//     PlcTask Inputs/GVL_iXlinker.EtherCAT_Master_EPPxxxx.Beckhoff_EPP6xxx.Beckhoff_EPP6xxxEK1122.A_0002_EPP6001_0002_0017.COM_Inputs.Data_In[11] <-> COM Inputs/Data In 11
//     PlcTask Inputs/GVL_iXlinker.EtherCAT_Master_EPPxxxx.Beckhoff_EPP6xxx.Beckhoff_EPP6xxxEK1122.A_0002_EPP6001_0002_0017.COM_Inputs.Data_In[12] <-> COM Inputs/Data In 12
//     PlcTask Inputs/GVL_iXlinker.EtherCAT_Master_EPPxxxx.Beckhoff_EPP6xxx.Beckhoff_EPP6xxxEK1122.A_0002_EPP6001_0002_0017.COM_Inputs.Data_In[13] <-> COM Inputs/Data In 13
//     PlcTask Inputs/GVL_iXlinker.EtherCAT_Master_EPPxxxx.Beckhoff_EPP6xxx.Beckhoff_EPP6xxxEK1122.A_0002_EPP6001_0002_0017.COM_Inputs.Data_In[14] <-> COM Inputs/Data In 14
//     PlcTask Inputs/GVL_iXlinker.EtherCAT_Master_EPPxxxx.Beckhoff_EPP6xxx.Beckhoff_EPP6xxxEK1122.A_0002_EPP6001_0002_0017.COM_Inputs.Data_In[15] <-> COM Inputs/Data In 15
//     PlcTask Inputs/GVL_iXlinker.EtherCAT_Master_EPPxxxx.Beckhoff_EPP6xxx.Beckhoff_EPP6xxxEK1122.A_0002_EPP6001_0002_0017.COM_Inputs.Data_In[16] <-> COM Inputs/Data In 16
//     PlcTask Inputs/GVL_iXlinker.EtherCAT_Master_EPPxxxx.Beckhoff_EPP6xxx.Beckhoff_EPP6xxxEK1122.A_0002_EPP6001_0002_0017.COM_Inputs.Data_In[17] <-> COM Inputs/Data In 17
//     PlcTask Inputs/GVL_iXlinker.EtherCAT_Master_EPPxxxx.Beckhoff_EPP6xxx.Beckhoff_EPP6xxxEK1122.A_0002_EPP6001_0002_0017.COM_Inputs.Data_In[18] <-> COM Inputs/Data In 18
//     PlcTask Inputs/GVL_iXlinker.EtherCAT_Master_EPPxxxx.Beckhoff_EPP6xxx.Beckhoff_EPP6xxxEK1122.A_0002_EPP6001_0002_0017.COM_Inputs.Data_In[19] <-> COM Inputs/Data In 19
//     PlcTask Inputs/GVL_iXlinker.EtherCAT_Master_EPPxxxx.Beckhoff_EPP6xxx.Beckhoff_EPP6xxxEK1122.A_0002_EPP6001_0002_0017.COM_Inputs.Data_In[20] <-> COM Inputs/Data In 20
//     PlcTask Inputs/GVL_iXlinker.EtherCAT_Master_EPPxxxx.Beckhoff_EPP6xxx.Beckhoff_EPP6xxxEK1122.A_0002_EPP6001_0002_0017.COM_Inputs.Data_In[21] <-> COM Inputs/Data In 21
//     PlcTask Outputs/GVL_iXlinker.EtherCAT_Master_EPPxxxx.Beckhoff_EPP6xxx.Beckhoff_EPP6xxxEK1122.A_0002_EPP6001_0002_0017.COM_Outputs.Ctrl <-> COM Outputs/Ctrl
//     PlcTask Outputs/GVL_iXlinker.EtherCAT_Master_EPPxxxx.Beckhoff_EPP6xxx.Beckhoff_EPP6xxxEK1122.A_0002_EPP6001_0002_0017.COM_Outputs.Data_Out[0] <-> COM Outputs/Data Out 0
//     PlcTask Outputs/GVL_iXlinker.EtherCAT_Master_EPPxxxx.Beckhoff_EPP6xxx.Beckhoff_EPP6xxxEK1122.A_0002_EPP6001_0002_0017.COM_Outputs.Data_Out[1] <-> COM Outputs/Data Out 1
//     PlcTask Outputs/GVL_iXlinker.EtherCAT_Master_EPPxxxx.Beckhoff_EPP6xxx.Beckhoff_EPP6xxxEK1122.A_0002_EPP6001_0002_0017.COM_Outputs.Data_Out[2] <-> COM Outputs/Data Out 2
//     PlcTask Outputs/GVL_iXlinker.EtherCAT_Master_EPPxxxx.Beckhoff_EPP6xxx.Beckhoff_EPP6xxxEK1122.A_0002_EPP6001_0002_0017.COM_Outputs.Data_Out[3] <-> COM Outputs/Data Out 3
//     PlcTask Outputs/GVL_iXlinker.EtherCAT_Master_EPPxxxx.Beckhoff_EPP6xxx.Beckhoff_EPP6xxxEK1122.A_0002_EPP6001_0002_0017.COM_Outputs.Data_Out[4] <-> COM Outputs/Data Out 4
//     PlcTask Outputs/GVL_iXlinker.EtherCAT_Master_EPPxxxx.Beckhoff_EPP6xxx.Beckhoff_EPP6xxxEK1122.A_0002_EPP6001_0002_0017.COM_Outputs.Data_Out[5] <-> COM Outputs/Data Out 5
//     PlcTask Outputs/GVL_iXlinker.EtherCAT_Master_EPPxxxx.Beckhoff_EPP6xxx.Beckhoff_EPP6xxxEK1122.A_0002_EPP6001_0002_0017.COM_Outputs.Data_Out[6] <-> COM Outputs/Data Out 6
//     PlcTask Outputs/GVL_iXlinker.EtherCAT_Master_EPPxxxx.Beckhoff_EPP6xxx.Beckhoff_EPP6xxxEK1122.A_0002_EPP6001_0002_0017.COM_Outputs.Data_Out[7] <-> COM Outputs/Data Out 7
//     PlcTask Outputs/GVL_iXlinker.EtherCAT_Master_EPPxxxx.Beckhoff_EPP6xxx.Beckhoff_EPP6xxxEK1122.A_0002_EPP6001_0002_0017.COM_Outputs.Data_Out[8] <-> COM Outputs/Data Out 8
//     PlcTask Outputs/GVL_iXlinker.EtherCAT_Master_EPPxxxx.Beckhoff_EPP6xxx.Beckhoff_EPP6xxxEK1122.A_0002_EPP6001_0002_0017.COM_Outputs.Data_Out[9] <-> COM Outputs/Data Out 9
//     PlcTask Outputs/GVL_iXlinker.EtherCAT_Master_EPPxxxx.Beckhoff_EPP6xxx.Beckhoff_EPP6xxxEK1122.A_0002_EPP6001_0002_0017.COM_Outputs.Data_Out[10] <-> COM Outputs/Data Out 10
//     PlcTask Outputs/GVL_iXlinker.EtherCAT_Master_EPPxxxx.Beckhoff_EPP6xxx.Beckhoff_EPP6xxxEK1122.A_0002_EPP6001_0002_0017.COM_Outputs.Data_Out[11] <-> COM Outputs/Data Out 11
//     PlcTask Outputs/GVL_iXlinker.EtherCAT_Master_EPPxxxx.Beckhoff_EPP6xxx.Beckhoff_EPP6xxxEK1122.A_0002_EPP6001_0002_0017.COM_Outputs.Data_Out[12] <-> COM Outputs/Data Out 12
//     PlcTask Outputs/GVL_iXlinker.EtherCAT_Master_EPPxxxx.Beckhoff_EPP6xxx.Beckhoff_EPP6xxxEK1122.A_0002_EPP6001_0002_0017.COM_Outputs.Data_Out[13] <-> COM Outputs/Data Out 13
//     PlcTask Outputs/GVL_iXlinker.EtherCAT_Master_EPPxxxx.Beckhoff_EPP6xxx.Beckhoff_EPP6xxxEK1122.A_0002_EPP6001_0002_0017.COM_Outputs.Data_Out[14] <-> COM Outputs/Data Out 14
//     PlcTask Outputs/GVL_iXlinker.EtherCAT_Master_EPPxxxx.Beckhoff_EPP6xxx.Beckhoff_EPP6xxxEK1122.A_0002_EPP6001_0002_0017.COM_Outputs.Data_Out[15] <-> COM Outputs/Data Out 15
//     PlcTask Outputs/GVL_iXlinker.EtherCAT_Master_EPPxxxx.Beckhoff_EPP6xxx.Beckhoff_EPP6xxxEK1122.A_0002_EPP6001_0002_0017.COM_Outputs.Data_Out[16] <-> COM Outputs/Data Out 16
//     PlcTask Outputs/GVL_iXlinker.EtherCAT_Master_EPPxxxx.Beckhoff_EPP6xxx.Beckhoff_EPP6xxxEK1122.A_0002_EPP6001_0002_0017.COM_Outputs.Data_Out[17] <-> COM Outputs/Data Out 17
//     PlcTask Outputs/GVL_iXlinker.EtherCAT_Master_EPPxxxx.Beckhoff_EPP6xxx.Beckhoff_EPP6xxxEK1122.A_0002_EPP6001_0002_0017.COM_Outputs.Data_Out[18] <-> COM Outputs/Data Out 18
//     PlcTask Outputs/GVL_iXlinker.EtherCAT_Master_EPPxxxx.Beckhoff_EPP6xxx.Beckhoff_EPP6xxxEK1122.A_0002_EPP6001_0002_0017.COM_Outputs.Data_Out[19] <-> COM Outputs/Data Out 19
//     PlcTask Outputs/GVL_iXlinker.EtherCAT_Master_EPPxxxx.Beckhoff_EPP6xxx.Beckhoff_EPP6xxxEK1122.A_0002_EPP6001_0002_0017.COM_Outputs.Data_Out[20] <-> COM Outputs/Data Out 20
//     PlcTask Outputs/GVL_iXlinker.EtherCAT_Master_EPPxxxx.Beckhoff_EPP6xxx.Beckhoff_EPP6xxxEK1122.A_0002_EPP6001_0002_0017.COM_Outputs.Data_Out[21] <-> COM Outputs/Data Out 21
//     PlcTask Inputs/GVL_iXlinker.EtherCAT_Master_EPPxxxx.Beckhoff_EPP6xxx.Beckhoff_EPP6xxxEK1122.A_0002_EPP6001_0002_0017.WcState.WcState <-> WcState/WcState
//     PlcTask Inputs/GVL_iXlinker.EtherCAT_Master_EPPxxxx.Beckhoff_EPP6xxx.Beckhoff_EPP6xxxEK1122.A_0002_EPP6001_0002_0017.WcState.InputToggle <-> WcState/InputToggle
//     PlcTask Inputs/GVL_iXlinker.EtherCAT_Master_EPPxxxx.Beckhoff_EPP6xxx.Beckhoff_EPP6xxxEK1122.A_0002_EPP6001_0002_0017.InfoData.AdsAddr <-> InfoData/AdsAddr
//     PlcTask Inputs/GVL_iXlinker.EtherCAT_Master_EPPxxxx.Beckhoff_EPP6xxx.Beckhoff_EPP6xxxEK1122.A_0002_EPP6001_0002_0017.InfoData.State <-> InfoData/State
//   PLC/PLC Instance <-> EtherCAT Master EPPxxxx/Beckhoff EPP6xxx/Beckhoff EPP6xxxEK1122/A_0003(EPP6001-0002-0018)
//     PlcTask Inputs/GVL_iXlinker.EtherCAT_Master_EPPxxxx.Beckhoff_EPP6xxx.Beckhoff_EPP6xxxEK1122.A_0003_EPP6001_0002_0018.COM_Inputs.Status <-> COM Inputs/Status
//     PlcTask Inputs/GVL_iXlinker.EtherCAT_Master_EPPxxxx.Beckhoff_EPP6xxx.Beckhoff_EPP6xxxEK1122.A_0003_EPP6001_0002_0018.COM_Inputs.Data_In[0] <-> COM Inputs/Data In 0
//     PlcTask Inputs/GVL_iXlinker.EtherCAT_Master_EPPxxxx.Beckhoff_EPP6xxx.Beckhoff_EPP6xxxEK1122.A_0003_EPP6001_0002_0018.COM_Inputs.Data_In[1] <-> COM Inputs/Data In 1
//     PlcTask Inputs/GVL_iXlinker.EtherCAT_Master_EPPxxxx.Beckhoff_EPP6xxx.Beckhoff_EPP6xxxEK1122.A_0003_EPP6001_0002_0018.COM_Inputs.Data_In[2] <-> COM Inputs/Data In 2
//     PlcTask Inputs/GVL_iXlinker.EtherCAT_Master_EPPxxxx.Beckhoff_EPP6xxx.Beckhoff_EPP6xxxEK1122.A_0003_EPP6001_0002_0018.COM_Inputs.Data_In[3] <-> COM Inputs/Data In 3
//     PlcTask Inputs/GVL_iXlinker.EtherCAT_Master_EPPxxxx.Beckhoff_EPP6xxx.Beckhoff_EPP6xxxEK1122.A_0003_EPP6001_0002_0018.COM_Inputs.Data_In[4] <-> COM Inputs/Data In 4
//     PlcTask Inputs/GVL_iXlinker.EtherCAT_Master_EPPxxxx.Beckhoff_EPP6xxx.Beckhoff_EPP6xxxEK1122.A_0003_EPP6001_0002_0018.COM_Inputs.Data_In[5] <-> COM Inputs/Data In 5
//     PlcTask Inputs/GVL_iXlinker.EtherCAT_Master_EPPxxxx.Beckhoff_EPP6xxx.Beckhoff_EPP6xxxEK1122.A_0003_EPP6001_0002_0018.COM_Inputs.Data_In[6] <-> COM Inputs/Data In 6
//     PlcTask Inputs/GVL_iXlinker.EtherCAT_Master_EPPxxxx.Beckhoff_EPP6xxx.Beckhoff_EPP6xxxEK1122.A_0003_EPP6001_0002_0018.COM_Inputs.Data_In[7] <-> COM Inputs/Data In 7
//     PlcTask Inputs/GVL_iXlinker.EtherCAT_Master_EPPxxxx.Beckhoff_EPP6xxx.Beckhoff_EPP6xxxEK1122.A_0003_EPP6001_0002_0018.COM_Inputs.Data_In[8] <-> COM Inputs/Data In 8
//     PlcTask Inputs/GVL_iXlinker.EtherCAT_Master_EPPxxxx.Beckhoff_EPP6xxx.Beckhoff_EPP6xxxEK1122.A_0003_EPP6001_0002_0018.COM_Inputs.Data_In[9] <-> COM Inputs/Data In 9
//     PlcTask Inputs/GVL_iXlinker.EtherCAT_Master_EPPxxxx.Beckhoff_EPP6xxx.Beckhoff_EPP6xxxEK1122.A_0003_EPP6001_0002_0018.COM_Inputs.Data_In[10] <-> COM Inputs/Data In 10
//     PlcTask Inputs/GVL_iXlinker.EtherCAT_Master_EPPxxxx.Beckhoff_EPP6xxx.Beckhoff_EPP6xxxEK1122.A_0003_EPP6001_0002_0018.COM_Inputs.Data_In[11] <-> COM Inputs/Data In 11
//     PlcTask Inputs/GVL_iXlinker.EtherCAT_Master_EPPxxxx.Beckhoff_EPP6xxx.Beckhoff_EPP6xxxEK1122.A_0003_EPP6001_0002_0018.COM_Inputs.Data_In[12] <-> COM Inputs/Data In 12
//     PlcTask Inputs/GVL_iXlinker.EtherCAT_Master_EPPxxxx.Beckhoff_EPP6xxx.Beckhoff_EPP6xxxEK1122.A_0003_EPP6001_0002_0018.COM_Inputs.Data_In[13] <-> COM Inputs/Data In 13
//     PlcTask Inputs/GVL_iXlinker.EtherCAT_Master_EPPxxxx.Beckhoff_EPP6xxx.Beckhoff_EPP6xxxEK1122.A_0003_EPP6001_0002_0018.COM_Inputs.Data_In[14] <-> COM Inputs/Data In 14
//     PlcTask Inputs/GVL_iXlinker.EtherCAT_Master_EPPxxxx.Beckhoff_EPP6xxx.Beckhoff_EPP6xxxEK1122.A_0003_EPP6001_0002_0018.COM_Inputs.Data_In[15] <-> COM Inputs/Data In 15
//     PlcTask Inputs/GVL_iXlinker.EtherCAT_Master_EPPxxxx.Beckhoff_EPP6xxx.Beckhoff_EPP6xxxEK1122.A_0003_EPP6001_0002_0018.COM_Inputs.Data_In[16] <-> COM Inputs/Data In 16
//     PlcTask Inputs/GVL_iXlinker.EtherCAT_Master_EPPxxxx.Beckhoff_EPP6xxx.Beckhoff_EPP6xxxEK1122.A_0003_EPP6001_0002_0018.COM_Inputs.Data_In[17] <-> COM Inputs/Data In 17
//     PlcTask Inputs/GVL_iXlinker.EtherCAT_Master_EPPxxxx.Beckhoff_EPP6xxx.Beckhoff_EPP6xxxEK1122.A_0003_EPP6001_0002_0018.COM_Inputs.Data_In[18] <-> COM Inputs/Data In 18
//     PlcTask Inputs/GVL_iXlinker.EtherCAT_Master_EPPxxxx.Beckhoff_EPP6xxx.Beckhoff_EPP6xxxEK1122.A_0003_EPP6001_0002_0018.COM_Inputs.Data_In[19] <-> COM Inputs/Data In 19
//     PlcTask Inputs/GVL_iXlinker.EtherCAT_Master_EPPxxxx.Beckhoff_EPP6xxx.Beckhoff_EPP6xxxEK1122.A_0003_EPP6001_0002_0018.COM_Inputs.Data_In[20] <-> COM Inputs/Data In 20
//     PlcTask Inputs/GVL_iXlinker.EtherCAT_Master_EPPxxxx.Beckhoff_EPP6xxx.Beckhoff_EPP6xxxEK1122.A_0003_EPP6001_0002_0018.COM_Inputs.Data_In[21] <-> COM Inputs/Data In 21
//     PlcTask Outputs/GVL_iXlinker.EtherCAT_Master_EPPxxxx.Beckhoff_EPP6xxx.Beckhoff_EPP6xxxEK1122.A_0003_EPP6001_0002_0018.COM_Outputs.Ctrl <-> COM Outputs/Ctrl
//     PlcTask Outputs/GVL_iXlinker.EtherCAT_Master_EPPxxxx.Beckhoff_EPP6xxx.Beckhoff_EPP6xxxEK1122.A_0003_EPP6001_0002_0018.COM_Outputs.Data_Out[0] <-> COM Outputs/Data Out 0
//     PlcTask Outputs/GVL_iXlinker.EtherCAT_Master_EPPxxxx.Beckhoff_EPP6xxx.Beckhoff_EPP6xxxEK1122.A_0003_EPP6001_0002_0018.COM_Outputs.Data_Out[1] <-> COM Outputs/Data Out 1
//     PlcTask Outputs/GVL_iXlinker.EtherCAT_Master_EPPxxxx.Beckhoff_EPP6xxx.Beckhoff_EPP6xxxEK1122.A_0003_EPP6001_0002_0018.COM_Outputs.Data_Out[2] <-> COM Outputs/Data Out 2
//     PlcTask Outputs/GVL_iXlinker.EtherCAT_Master_EPPxxxx.Beckhoff_EPP6xxx.Beckhoff_EPP6xxxEK1122.A_0003_EPP6001_0002_0018.COM_Outputs.Data_Out[3] <-> COM Outputs/Data Out 3
//     PlcTask Outputs/GVL_iXlinker.EtherCAT_Master_EPPxxxx.Beckhoff_EPP6xxx.Beckhoff_EPP6xxxEK1122.A_0003_EPP6001_0002_0018.COM_Outputs.Data_Out[4] <-> COM Outputs/Data Out 4
//     PlcTask Outputs/GVL_iXlinker.EtherCAT_Master_EPPxxxx.Beckhoff_EPP6xxx.Beckhoff_EPP6xxxEK1122.A_0003_EPP6001_0002_0018.COM_Outputs.Data_Out[5] <-> COM Outputs/Data Out 5
//     PlcTask Outputs/GVL_iXlinker.EtherCAT_Master_EPPxxxx.Beckhoff_EPP6xxx.Beckhoff_EPP6xxxEK1122.A_0003_EPP6001_0002_0018.COM_Outputs.Data_Out[6] <-> COM Outputs/Data Out 6
//     PlcTask Outputs/GVL_iXlinker.EtherCAT_Master_EPPxxxx.Beckhoff_EPP6xxx.Beckhoff_EPP6xxxEK1122.A_0003_EPP6001_0002_0018.COM_Outputs.Data_Out[7] <-> COM Outputs/Data Out 7
//     PlcTask Outputs/GVL_iXlinker.EtherCAT_Master_EPPxxxx.Beckhoff_EPP6xxx.Beckhoff_EPP6xxxEK1122.A_0003_EPP6001_0002_0018.COM_Outputs.Data_Out[8] <-> COM Outputs/Data Out 8
//     PlcTask Outputs/GVL_iXlinker.EtherCAT_Master_EPPxxxx.Beckhoff_EPP6xxx.Beckhoff_EPP6xxxEK1122.A_0003_EPP6001_0002_0018.COM_Outputs.Data_Out[9] <-> COM Outputs/Data Out 9
//     PlcTask Outputs/GVL_iXlinker.EtherCAT_Master_EPPxxxx.Beckhoff_EPP6xxx.Beckhoff_EPP6xxxEK1122.A_0003_EPP6001_0002_0018.COM_Outputs.Data_Out[10] <-> COM Outputs/Data Out 10
//     PlcTask Outputs/GVL_iXlinker.EtherCAT_Master_EPPxxxx.Beckhoff_EPP6xxx.Beckhoff_EPP6xxxEK1122.A_0003_EPP6001_0002_0018.COM_Outputs.Data_Out[11] <-> COM Outputs/Data Out 11
//     PlcTask Outputs/GVL_iXlinker.EtherCAT_Master_EPPxxxx.Beckhoff_EPP6xxx.Beckhoff_EPP6xxxEK1122.A_0003_EPP6001_0002_0018.COM_Outputs.Data_Out[12] <-> COM Outputs/Data Out 12
//     PlcTask Outputs/GVL_iXlinker.EtherCAT_Master_EPPxxxx.Beckhoff_EPP6xxx.Beckhoff_EPP6xxxEK1122.A_0003_EPP6001_0002_0018.COM_Outputs.Data_Out[13] <-> COM Outputs/Data Out 13
//     PlcTask Outputs/GVL_iXlinker.EtherCAT_Master_EPPxxxx.Beckhoff_EPP6xxx.Beckhoff_EPP6xxxEK1122.A_0003_EPP6001_0002_0018.COM_Outputs.Data_Out[14] <-> COM Outputs/Data Out 14
//     PlcTask Outputs/GVL_iXlinker.EtherCAT_Master_EPPxxxx.Beckhoff_EPP6xxx.Beckhoff_EPP6xxxEK1122.A_0003_EPP6001_0002_0018.COM_Outputs.Data_Out[15] <-> COM Outputs/Data Out 15
//     PlcTask Outputs/GVL_iXlinker.EtherCAT_Master_EPPxxxx.Beckhoff_EPP6xxx.Beckhoff_EPP6xxxEK1122.A_0003_EPP6001_0002_0018.COM_Outputs.Data_Out[16] <-> COM Outputs/Data Out 16
//     PlcTask Outputs/GVL_iXlinker.EtherCAT_Master_EPPxxxx.Beckhoff_EPP6xxx.Beckhoff_EPP6xxxEK1122.A_0003_EPP6001_0002_0018.COM_Outputs.Data_Out[17] <-> COM Outputs/Data Out 17
//     PlcTask Outputs/GVL_iXlinker.EtherCAT_Master_EPPxxxx.Beckhoff_EPP6xxx.Beckhoff_EPP6xxxEK1122.A_0003_EPP6001_0002_0018.COM_Outputs.Data_Out[18] <-> COM Outputs/Data Out 18
//     PlcTask Outputs/GVL_iXlinker.EtherCAT_Master_EPPxxxx.Beckhoff_EPP6xxx.Beckhoff_EPP6xxxEK1122.A_0003_EPP6001_0002_0018.COM_Outputs.Data_Out[19] <-> COM Outputs/Data Out 19
//     PlcTask Outputs/GVL_iXlinker.EtherCAT_Master_EPPxxxx.Beckhoff_EPP6xxx.Beckhoff_EPP6xxxEK1122.A_0003_EPP6001_0002_0018.COM_Outputs.Data_Out[20] <-> COM Outputs/Data Out 20
//     PlcTask Outputs/GVL_iXlinker.EtherCAT_Master_EPPxxxx.Beckhoff_EPP6xxx.Beckhoff_EPP6xxxEK1122.A_0003_EPP6001_0002_0018.COM_Outputs.Data_Out[21] <-> COM Outputs/Data Out 21
//     PlcTask Inputs/GVL_iXlinker.EtherCAT_Master_EPPxxxx.Beckhoff_EPP6xxx.Beckhoff_EPP6xxxEK1122.A_0003_EPP6001_0002_0018.WcState.WcState <-> WcState/WcState
//     PlcTask Inputs/GVL_iXlinker.EtherCAT_Master_EPPxxxx.Beckhoff_EPP6xxx.Beckhoff_EPP6xxxEK1122.A_0003_EPP6001_0002_0018.WcState.InputToggle <-> WcState/InputToggle
//     PlcTask Inputs/GVL_iXlinker.EtherCAT_Master_EPPxxxx.Beckhoff_EPP6xxx.Beckhoff_EPP6xxxEK1122.A_0003_EPP6001_0002_0018.InfoData.AdsAddr <-> InfoData/AdsAddr
//     PlcTask Inputs/GVL_iXlinker.EtherCAT_Master_EPPxxxx.Beckhoff_EPP6xxx.Beckhoff_EPP6xxxEK1122.A_0003_EPP6001_0002_0018.InfoData.State <-> InfoData/State
//   PLC/PLC Instance <-> EtherCAT Master EPPxxxx/Beckhoff EPP6xxx/Beckhoff EPP6xxxEK1122/A_0004(EPP6002-0002-0016)
//     PlcTask Inputs/GVL_iXlinker.EtherCAT_Master_EPPxxxx.Beckhoff_EPP6xxx.Beckhoff_EPP6xxxEK1122.A_0004_EPP6002_0002_0016.COM_TxPDO_Map_Inputs_Channel_1.Status <-> COM TxPDO-Map Inputs Channel 1/Status
//     PlcTask Inputs/GVL_iXlinker.EtherCAT_Master_EPPxxxx.Beckhoff_EPP6xxx.Beckhoff_EPP6xxxEK1122.A_0004_EPP6002_0002_0016.COM_TxPDO_Map_Inputs_Channel_2.Status <-> COM TxPDO-Map Inputs Channel 2/Status
//     PlcTask Inputs/GVL_iXlinker.EtherCAT_Master_EPPxxxx.Beckhoff_EPP6xxx.Beckhoff_EPP6xxxEK1122.A_0004_EPP6002_0002_0016.COM_TxPDO_Map_Inputs_Channel_1.Data_In[0] <-> COM TxPDO-Map Inputs Channel 1/Data In 0
//     PlcTask Inputs/GVL_iXlinker.EtherCAT_Master_EPPxxxx.Beckhoff_EPP6xxx.Beckhoff_EPP6xxxEK1122.A_0004_EPP6002_0002_0016.COM_TxPDO_Map_Inputs_Channel_1.Data_In[1] <-> COM TxPDO-Map Inputs Channel 1/Data In 1
//     PlcTask Inputs/GVL_iXlinker.EtherCAT_Master_EPPxxxx.Beckhoff_EPP6xxx.Beckhoff_EPP6xxxEK1122.A_0004_EPP6002_0002_0016.COM_TxPDO_Map_Inputs_Channel_1.Data_In[2] <-> COM TxPDO-Map Inputs Channel 1/Data In 2
//     PlcTask Inputs/GVL_iXlinker.EtherCAT_Master_EPPxxxx.Beckhoff_EPP6xxx.Beckhoff_EPP6xxxEK1122.A_0004_EPP6002_0002_0016.COM_TxPDO_Map_Inputs_Channel_1.Data_In[3] <-> COM TxPDO-Map Inputs Channel 1/Data In 3
//     PlcTask Inputs/GVL_iXlinker.EtherCAT_Master_EPPxxxx.Beckhoff_EPP6xxx.Beckhoff_EPP6xxxEK1122.A_0004_EPP6002_0002_0016.COM_TxPDO_Map_Inputs_Channel_1.Data_In[4] <-> COM TxPDO-Map Inputs Channel 1/Data In 4
//     PlcTask Inputs/GVL_iXlinker.EtherCAT_Master_EPPxxxx.Beckhoff_EPP6xxx.Beckhoff_EPP6xxxEK1122.A_0004_EPP6002_0002_0016.COM_TxPDO_Map_Inputs_Channel_1.Data_In[5] <-> COM TxPDO-Map Inputs Channel 1/Data In 5
//     PlcTask Inputs/GVL_iXlinker.EtherCAT_Master_EPPxxxx.Beckhoff_EPP6xxx.Beckhoff_EPP6xxxEK1122.A_0004_EPP6002_0002_0016.COM_TxPDO_Map_Inputs_Channel_1.Data_In[6] <-> COM TxPDO-Map Inputs Channel 1/Data In 6
//     PlcTask Inputs/GVL_iXlinker.EtherCAT_Master_EPPxxxx.Beckhoff_EPP6xxx.Beckhoff_EPP6xxxEK1122.A_0004_EPP6002_0002_0016.COM_TxPDO_Map_Inputs_Channel_1.Data_In[7] <-> COM TxPDO-Map Inputs Channel 1/Data In 7
//     PlcTask Inputs/GVL_iXlinker.EtherCAT_Master_EPPxxxx.Beckhoff_EPP6xxx.Beckhoff_EPP6xxxEK1122.A_0004_EPP6002_0002_0016.COM_TxPDO_Map_Inputs_Channel_1.Data_In[8] <-> COM TxPDO-Map Inputs Channel 1/Data In 8
//     PlcTask Inputs/GVL_iXlinker.EtherCAT_Master_EPPxxxx.Beckhoff_EPP6xxx.Beckhoff_EPP6xxxEK1122.A_0004_EPP6002_0002_0016.COM_TxPDO_Map_Inputs_Channel_1.Data_In[9] <-> COM TxPDO-Map Inputs Channel 1/Data In 9
//     PlcTask Inputs/GVL_iXlinker.EtherCAT_Master_EPPxxxx.Beckhoff_EPP6xxx.Beckhoff_EPP6xxxEK1122.A_0004_EPP6002_0002_0016.COM_TxPDO_Map_Inputs_Channel_1.Data_In[10] <-> COM TxPDO-Map Inputs Channel 1/Data In 10
//     PlcTask Inputs/GVL_iXlinker.EtherCAT_Master_EPPxxxx.Beckhoff_EPP6xxx.Beckhoff_EPP6xxxEK1122.A_0004_EPP6002_0002_0016.COM_TxPDO_Map_Inputs_Channel_1.Data_In[11] <-> COM TxPDO-Map Inputs Channel 1/Data In 11
//     PlcTask Inputs/GVL_iXlinker.EtherCAT_Master_EPPxxxx.Beckhoff_EPP6xxx.Beckhoff_EPP6xxxEK1122.A_0004_EPP6002_0002_0016.COM_TxPDO_Map_Inputs_Channel_1.Data_In[12] <-> COM TxPDO-Map Inputs Channel 1/Data In 12
//     PlcTask Inputs/GVL_iXlinker.EtherCAT_Master_EPPxxxx.Beckhoff_EPP6xxx.Beckhoff_EPP6xxxEK1122.A_0004_EPP6002_0002_0016.COM_TxPDO_Map_Inputs_Channel_1.Data_In[13] <-> COM TxPDO-Map Inputs Channel 1/Data In 13
//     PlcTask Inputs/GVL_iXlinker.EtherCAT_Master_EPPxxxx.Beckhoff_EPP6xxx.Beckhoff_EPP6xxxEK1122.A_0004_EPP6002_0002_0016.COM_TxPDO_Map_Inputs_Channel_1.Data_In[14] <-> COM TxPDO-Map Inputs Channel 1/Data In 14
//     PlcTask Inputs/GVL_iXlinker.EtherCAT_Master_EPPxxxx.Beckhoff_EPP6xxx.Beckhoff_EPP6xxxEK1122.A_0004_EPP6002_0002_0016.COM_TxPDO_Map_Inputs_Channel_1.Data_In[15] <-> COM TxPDO-Map Inputs Channel 1/Data In 15
//     PlcTask Inputs/GVL_iXlinker.EtherCAT_Master_EPPxxxx.Beckhoff_EPP6xxx.Beckhoff_EPP6xxxEK1122.A_0004_EPP6002_0002_0016.COM_TxPDO_Map_Inputs_Channel_1.Data_In[16] <-> COM TxPDO-Map Inputs Channel 1/Data In 16
//     PlcTask Inputs/GVL_iXlinker.EtherCAT_Master_EPPxxxx.Beckhoff_EPP6xxx.Beckhoff_EPP6xxxEK1122.A_0004_EPP6002_0002_0016.COM_TxPDO_Map_Inputs_Channel_1.Data_In[17] <-> COM TxPDO-Map Inputs Channel 1/Data In 17
//     PlcTask Inputs/GVL_iXlinker.EtherCAT_Master_EPPxxxx.Beckhoff_EPP6xxx.Beckhoff_EPP6xxxEK1122.A_0004_EPP6002_0002_0016.COM_TxPDO_Map_Inputs_Channel_1.Data_In[18] <-> COM TxPDO-Map Inputs Channel 1/Data In 18
//     PlcTask Inputs/GVL_iXlinker.EtherCAT_Master_EPPxxxx.Beckhoff_EPP6xxx.Beckhoff_EPP6xxxEK1122.A_0004_EPP6002_0002_0016.COM_TxPDO_Map_Inputs_Channel_1.Data_In[19] <-> COM TxPDO-Map Inputs Channel 1/Data In 19
//     PlcTask Inputs/GVL_iXlinker.EtherCAT_Master_EPPxxxx.Beckhoff_EPP6xxx.Beckhoff_EPP6xxxEK1122.A_0004_EPP6002_0002_0016.COM_TxPDO_Map_Inputs_Channel_1.Data_In[20] <-> COM TxPDO-Map Inputs Channel 1/Data In 20
//     PlcTask Inputs/GVL_iXlinker.EtherCAT_Master_EPPxxxx.Beckhoff_EPP6xxx.Beckhoff_EPP6xxxEK1122.A_0004_EPP6002_0002_0016.COM_TxPDO_Map_Inputs_Channel_1.Data_In[21] <-> COM TxPDO-Map Inputs Channel 1/Data In 21
//     PlcTask Inputs/GVL_iXlinker.EtherCAT_Master_EPPxxxx.Beckhoff_EPP6xxx.Beckhoff_EPP6xxxEK1122.A_0004_EPP6002_0002_0016.COM_TxPDO_Map_Inputs_Channel_2.Data_In[0] <-> COM TxPDO-Map Inputs Channel 2/Data In 0
//     PlcTask Inputs/GVL_iXlinker.EtherCAT_Master_EPPxxxx.Beckhoff_EPP6xxx.Beckhoff_EPP6xxxEK1122.A_0004_EPP6002_0002_0016.COM_TxPDO_Map_Inputs_Channel_2.Data_In[1] <-> COM TxPDO-Map Inputs Channel 2/Data In 1
//     PlcTask Inputs/GVL_iXlinker.EtherCAT_Master_EPPxxxx.Beckhoff_EPP6xxx.Beckhoff_EPP6xxxEK1122.A_0004_EPP6002_0002_0016.COM_TxPDO_Map_Inputs_Channel_2.Data_In[2] <-> COM TxPDO-Map Inputs Channel 2/Data In 2
//     PlcTask Inputs/GVL_iXlinker.EtherCAT_Master_EPPxxxx.Beckhoff_EPP6xxx.Beckhoff_EPP6xxxEK1122.A_0004_EPP6002_0002_0016.COM_TxPDO_Map_Inputs_Channel_2.Data_In[3] <-> COM TxPDO-Map Inputs Channel 2/Data In 3
//     PlcTask Inputs/GVL_iXlinker.EtherCAT_Master_EPPxxxx.Beckhoff_EPP6xxx.Beckhoff_EPP6xxxEK1122.A_0004_EPP6002_0002_0016.COM_TxPDO_Map_Inputs_Channel_2.Data_In[4] <-> COM TxPDO-Map Inputs Channel 2/Data In 4
//     PlcTask Inputs/GVL_iXlinker.EtherCAT_Master_EPPxxxx.Beckhoff_EPP6xxx.Beckhoff_EPP6xxxEK1122.A_0004_EPP6002_0002_0016.COM_TxPDO_Map_Inputs_Channel_2.Data_In[5] <-> COM TxPDO-Map Inputs Channel 2/Data In 5
//     PlcTask Inputs/GVL_iXlinker.EtherCAT_Master_EPPxxxx.Beckhoff_EPP6xxx.Beckhoff_EPP6xxxEK1122.A_0004_EPP6002_0002_0016.COM_TxPDO_Map_Inputs_Channel_2.Data_In[6] <-> COM TxPDO-Map Inputs Channel 2/Data In 6
//     PlcTask Inputs/GVL_iXlinker.EtherCAT_Master_EPPxxxx.Beckhoff_EPP6xxx.Beckhoff_EPP6xxxEK1122.A_0004_EPP6002_0002_0016.COM_TxPDO_Map_Inputs_Channel_2.Data_In[7] <-> COM TxPDO-Map Inputs Channel 2/Data In 7
//     PlcTask Inputs/GVL_iXlinker.EtherCAT_Master_EPPxxxx.Beckhoff_EPP6xxx.Beckhoff_EPP6xxxEK1122.A_0004_EPP6002_0002_0016.COM_TxPDO_Map_Inputs_Channel_2.Data_In[8] <-> COM TxPDO-Map Inputs Channel 2/Data In 8
//     PlcTask Inputs/GVL_iXlinker.EtherCAT_Master_EPPxxxx.Beckhoff_EPP6xxx.Beckhoff_EPP6xxxEK1122.A_0004_EPP6002_0002_0016.COM_TxPDO_Map_Inputs_Channel_2.Data_In[9] <-> COM TxPDO-Map Inputs Channel 2/Data In 9
//     PlcTask Inputs/GVL_iXlinker.EtherCAT_Master_EPPxxxx.Beckhoff_EPP6xxx.Beckhoff_EPP6xxxEK1122.A_0004_EPP6002_0002_0016.COM_TxPDO_Map_Inputs_Channel_2.Data_In[10] <-> COM TxPDO-Map Inputs Channel 2/Data In 10
//     PlcTask Inputs/GVL_iXlinker.EtherCAT_Master_EPPxxxx.Beckhoff_EPP6xxx.Beckhoff_EPP6xxxEK1122.A_0004_EPP6002_0002_0016.COM_TxPDO_Map_Inputs_Channel_2.Data_In[11] <-> COM TxPDO-Map Inputs Channel 2/Data In 11
//     PlcTask Inputs/GVL_iXlinker.EtherCAT_Master_EPPxxxx.Beckhoff_EPP6xxx.Beckhoff_EPP6xxxEK1122.A_0004_EPP6002_0002_0016.COM_TxPDO_Map_Inputs_Channel_2.Data_In[12] <-> COM TxPDO-Map Inputs Channel 2/Data In 12
//     PlcTask Inputs/GVL_iXlinker.EtherCAT_Master_EPPxxxx.Beckhoff_EPP6xxx.Beckhoff_EPP6xxxEK1122.A_0004_EPP6002_0002_0016.COM_TxPDO_Map_Inputs_Channel_2.Data_In[13] <-> COM TxPDO-Map Inputs Channel 2/Data In 13
//     PlcTask Inputs/GVL_iXlinker.EtherCAT_Master_EPPxxxx.Beckhoff_EPP6xxx.Beckhoff_EPP6xxxEK1122.A_0004_EPP6002_0002_0016.COM_TxPDO_Map_Inputs_Channel_2.Data_In[14] <-> COM TxPDO-Map Inputs Channel 2/Data In 14
//     PlcTask Inputs/GVL_iXlinker.EtherCAT_Master_EPPxxxx.Beckhoff_EPP6xxx.Beckhoff_EPP6xxxEK1122.A_0004_EPP6002_0002_0016.COM_TxPDO_Map_Inputs_Channel_2.Data_In[15] <-> COM TxPDO-Map Inputs Channel 2/Data In 15
//     PlcTask Inputs/GVL_iXlinker.EtherCAT_Master_EPPxxxx.Beckhoff_EPP6xxx.Beckhoff_EPP6xxxEK1122.A_0004_EPP6002_0002_0016.COM_TxPDO_Map_Inputs_Channel_2.Data_In[16] <-> COM TxPDO-Map Inputs Channel 2/Data In 16
//     PlcTask Inputs/GVL_iXlinker.EtherCAT_Master_EPPxxxx.Beckhoff_EPP6xxx.Beckhoff_EPP6xxxEK1122.A_0004_EPP6002_0002_0016.COM_TxPDO_Map_Inputs_Channel_2.Data_In[17] <-> COM TxPDO-Map Inputs Channel 2/Data In 17
//     PlcTask Inputs/GVL_iXlinker.EtherCAT_Master_EPPxxxx.Beckhoff_EPP6xxx.Beckhoff_EPP6xxxEK1122.A_0004_EPP6002_0002_0016.COM_TxPDO_Map_Inputs_Channel_2.Data_In[18] <-> COM TxPDO-Map Inputs Channel 2/Data In 18
//     PlcTask Inputs/GVL_iXlinker.EtherCAT_Master_EPPxxxx.Beckhoff_EPP6xxx.Beckhoff_EPP6xxxEK1122.A_0004_EPP6002_0002_0016.COM_TxPDO_Map_Inputs_Channel_2.Data_In[19] <-> COM TxPDO-Map Inputs Channel 2/Data In 19
//     PlcTask Inputs/GVL_iXlinker.EtherCAT_Master_EPPxxxx.Beckhoff_EPP6xxx.Beckhoff_EPP6xxxEK1122.A_0004_EPP6002_0002_0016.COM_TxPDO_Map_Inputs_Channel_2.Data_In[20] <-> COM TxPDO-Map Inputs Channel 2/Data In 20
//     PlcTask Inputs/GVL_iXlinker.EtherCAT_Master_EPPxxxx.Beckhoff_EPP6xxx.Beckhoff_EPP6xxxEK1122.A_0004_EPP6002_0002_0016.COM_TxPDO_Map_Inputs_Channel_2.Data_In[21] <-> COM TxPDO-Map Inputs Channel 2/Data In 21
//     PlcTask Outputs/GVL_iXlinker.EtherCAT_Master_EPPxxxx.Beckhoff_EPP6xxx.Beckhoff_EPP6xxxEK1122.A_0004_EPP6002_0002_0016.COM_RxPDO_Map_Outputs_Channel_1.Ctrl <-> COM RxPDO-Map Outputs Channel 1/Ctrl
//     PlcTask Outputs/GVL_iXlinker.EtherCAT_Master_EPPxxxx.Beckhoff_EPP6xxx.Beckhoff_EPP6xxxEK1122.A_0004_EPP6002_0002_0016.COM_RxPDO_Map_Outputs_Channel_2.Ctrl <-> COM RxPDO-Map Outputs Channel 2/Ctrl
//     PlcTask Outputs/GVL_iXlinker.EtherCAT_Master_EPPxxxx.Beckhoff_EPP6xxx.Beckhoff_EPP6xxxEK1122.A_0004_EPP6002_0002_0016.COM_RxPDO_Map_Outputs_Channel_1.Data_Out[0] <-> COM RxPDO-Map Outputs Channel 1/Data Out 0
//     PlcTask Outputs/GVL_iXlinker.EtherCAT_Master_EPPxxxx.Beckhoff_EPP6xxx.Beckhoff_EPP6xxxEK1122.A_0004_EPP6002_0002_0016.COM_RxPDO_Map_Outputs_Channel_1.Data_Out[1] <-> COM RxPDO-Map Outputs Channel 1/Data Out 1
//     PlcTask Outputs/GVL_iXlinker.EtherCAT_Master_EPPxxxx.Beckhoff_EPP6xxx.Beckhoff_EPP6xxxEK1122.A_0004_EPP6002_0002_0016.COM_RxPDO_Map_Outputs_Channel_1.Data_Out[2] <-> COM RxPDO-Map Outputs Channel 1/Data Out 2
//     PlcTask Outputs/GVL_iXlinker.EtherCAT_Master_EPPxxxx.Beckhoff_EPP6xxx.Beckhoff_EPP6xxxEK1122.A_0004_EPP6002_0002_0016.COM_RxPDO_Map_Outputs_Channel_1.Data_Out[3] <-> COM RxPDO-Map Outputs Channel 1/Data Out 3
//     PlcTask Outputs/GVL_iXlinker.EtherCAT_Master_EPPxxxx.Beckhoff_EPP6xxx.Beckhoff_EPP6xxxEK1122.A_0004_EPP6002_0002_0016.COM_RxPDO_Map_Outputs_Channel_1.Data_Out[4] <-> COM RxPDO-Map Outputs Channel 1/Data Out 4
//     PlcTask Outputs/GVL_iXlinker.EtherCAT_Master_EPPxxxx.Beckhoff_EPP6xxx.Beckhoff_EPP6xxxEK1122.A_0004_EPP6002_0002_0016.COM_RxPDO_Map_Outputs_Channel_1.Data_Out[5] <-> COM RxPDO-Map Outputs Channel 1/Data Out 5
//     PlcTask Outputs/GVL_iXlinker.EtherCAT_Master_EPPxxxx.Beckhoff_EPP6xxx.Beckhoff_EPP6xxxEK1122.A_0004_EPP6002_0002_0016.COM_RxPDO_Map_Outputs_Channel_1.Data_Out[6] <-> COM RxPDO-Map Outputs Channel 1/Data Out 6
//     PlcTask Outputs/GVL_iXlinker.EtherCAT_Master_EPPxxxx.Beckhoff_EPP6xxx.Beckhoff_EPP6xxxEK1122.A_0004_EPP6002_0002_0016.COM_RxPDO_Map_Outputs_Channel_1.Data_Out[7] <-> COM RxPDO-Map Outputs Channel 1/Data Out 7
//     PlcTask Outputs/GVL_iXlinker.EtherCAT_Master_EPPxxxx.Beckhoff_EPP6xxx.Beckhoff_EPP6xxxEK1122.A_0004_EPP6002_0002_0016.COM_RxPDO_Map_Outputs_Channel_1.Data_Out[8] <-> COM RxPDO-Map Outputs Channel 1/Data Out 8
//     PlcTask Outputs/GVL_iXlinker.EtherCAT_Master_EPPxxxx.Beckhoff_EPP6xxx.Beckhoff_EPP6xxxEK1122.A_0004_EPP6002_0002_0016.COM_RxPDO_Map_Outputs_Channel_1.Data_Out[9] <-> COM RxPDO-Map Outputs Channel 1/Data Out 9
//     PlcTask Outputs/GVL_iXlinker.EtherCAT_Master_EPPxxxx.Beckhoff_EPP6xxx.Beckhoff_EPP6xxxEK1122.A_0004_EPP6002_0002_0016.COM_RxPDO_Map_Outputs_Channel_1.Data_Out[10] <-> COM RxPDO-Map Outputs Channel 1/Data Out 10
//     PlcTask Outputs/GVL_iXlinker.EtherCAT_Master_EPPxxxx.Beckhoff_EPP6xxx.Beckhoff_EPP6xxxEK1122.A_0004_EPP6002_0002_0016.COM_RxPDO_Map_Outputs_Channel_1.Data_Out[11] <-> COM RxPDO-Map Outputs Channel 1/Data Out 11
//     PlcTask Outputs/GVL_iXlinker.EtherCAT_Master_EPPxxxx.Beckhoff_EPP6xxx.Beckhoff_EPP6xxxEK1122.A_0004_EPP6002_0002_0016.COM_RxPDO_Map_Outputs_Channel_1.Data_Out[12] <-> COM RxPDO-Map Outputs Channel 1/Data Out 12
//     PlcTask Outputs/GVL_iXlinker.EtherCAT_Master_EPPxxxx.Beckhoff_EPP6xxx.Beckhoff_EPP6xxxEK1122.A_0004_EPP6002_0002_0016.COM_RxPDO_Map_Outputs_Channel_1.Data_Out[13] <-> COM RxPDO-Map Outputs Channel 1/Data Out 13
//     PlcTask Outputs/GVL_iXlinker.EtherCAT_Master_EPPxxxx.Beckhoff_EPP6xxx.Beckhoff_EPP6xxxEK1122.A_0004_EPP6002_0002_0016.COM_RxPDO_Map_Outputs_Channel_1.Data_Out[14] <-> COM RxPDO-Map Outputs Channel 1/Data Out 14
//     PlcTask Outputs/GVL_iXlinker.EtherCAT_Master_EPPxxxx.Beckhoff_EPP6xxx.Beckhoff_EPP6xxxEK1122.A_0004_EPP6002_0002_0016.COM_RxPDO_Map_Outputs_Channel_1.Data_Out[15] <-> COM RxPDO-Map Outputs Channel 1/Data Out 15
//     PlcTask Outputs/GVL_iXlinker.EtherCAT_Master_EPPxxxx.Beckhoff_EPP6xxx.Beckhoff_EPP6xxxEK1122.A_0004_EPP6002_0002_0016.COM_RxPDO_Map_Outputs_Channel_1.Data_Out[16] <-> COM RxPDO-Map Outputs Channel 1/Data Out 16
//     PlcTask Outputs/GVL_iXlinker.EtherCAT_Master_EPPxxxx.Beckhoff_EPP6xxx.Beckhoff_EPP6xxxEK1122.A_0004_EPP6002_0002_0016.COM_RxPDO_Map_Outputs_Channel_1.Data_Out[17] <-> COM RxPDO-Map Outputs Channel 1/Data Out 17
//     PlcTask Outputs/GVL_iXlinker.EtherCAT_Master_EPPxxxx.Beckhoff_EPP6xxx.Beckhoff_EPP6xxxEK1122.A_0004_EPP6002_0002_0016.COM_RxPDO_Map_Outputs_Channel_1.Data_Out[18] <-> COM RxPDO-Map Outputs Channel 1/Data Out 18
//     PlcTask Outputs/GVL_iXlinker.EtherCAT_Master_EPPxxxx.Beckhoff_EPP6xxx.Beckhoff_EPP6xxxEK1122.A_0004_EPP6002_0002_0016.COM_RxPDO_Map_Outputs_Channel_1.Data_Out[19] <-> COM RxPDO-Map Outputs Channel 1/Data Out 19
//     PlcTask Outputs/GVL_iXlinker.EtherCAT_Master_EPPxxxx.Beckhoff_EPP6xxx.Beckhoff_EPP6xxxEK1122.A_0004_EPP6002_0002_0016.COM_RxPDO_Map_Outputs_Channel_1.Data_Out[20] <-> COM RxPDO-Map Outputs Channel 1/Data Out 20
//     PlcTask Outputs/GVL_iXlinker.EtherCAT_Master_EPPxxxx.Beckhoff_EPP6xxx.Beckhoff_EPP6xxxEK1122.A_0004_EPP6002_0002_0016.COM_RxPDO_Map_Outputs_Channel_1.Data_Out[21] <-> COM RxPDO-Map Outputs Channel 1/Data Out 21
//     PlcTask Outputs/GVL_iXlinker.EtherCAT_Master_EPPxxxx.Beckhoff_EPP6xxx.Beckhoff_EPP6xxxEK1122.A_0004_EPP6002_0002_0016.COM_RxPDO_Map_Outputs_Channel_2.Data_Out[0] <-> COM RxPDO-Map Outputs Channel 2/Data Out 0
//     PlcTask Outputs/GVL_iXlinker.EtherCAT_Master_EPPxxxx.Beckhoff_EPP6xxx.Beckhoff_EPP6xxxEK1122.A_0004_EPP6002_0002_0016.COM_RxPDO_Map_Outputs_Channel_2.Data_Out[1] <-> COM RxPDO-Map Outputs Channel 2/Data Out 1
//     PlcTask Outputs/GVL_iXlinker.EtherCAT_Master_EPPxxxx.Beckhoff_EPP6xxx.Beckhoff_EPP6xxxEK1122.A_0004_EPP6002_0002_0016.COM_RxPDO_Map_Outputs_Channel_2.Data_Out[2] <-> COM RxPDO-Map Outputs Channel 2/Data Out 2
//     PlcTask Outputs/GVL_iXlinker.EtherCAT_Master_EPPxxxx.Beckhoff_EPP6xxx.Beckhoff_EPP6xxxEK1122.A_0004_EPP6002_0002_0016.COM_RxPDO_Map_Outputs_Channel_2.Data_Out[3] <-> COM RxPDO-Map Outputs Channel 2/Data Out 3
//     PlcTask Outputs/GVL_iXlinker.EtherCAT_Master_EPPxxxx.Beckhoff_EPP6xxx.Beckhoff_EPP6xxxEK1122.A_0004_EPP6002_0002_0016.COM_RxPDO_Map_Outputs_Channel_2.Data_Out[4] <-> COM RxPDO-Map Outputs Channel 2/Data Out 4
//     PlcTask Outputs/GVL_iXlinker.EtherCAT_Master_EPPxxxx.Beckhoff_EPP6xxx.Beckhoff_EPP6xxxEK1122.A_0004_EPP6002_0002_0016.COM_RxPDO_Map_Outputs_Channel_2.Data_Out[5] <-> COM RxPDO-Map Outputs Channel 2/Data Out 5
//     PlcTask Outputs/GVL_iXlinker.EtherCAT_Master_EPPxxxx.Beckhoff_EPP6xxx.Beckhoff_EPP6xxxEK1122.A_0004_EPP6002_0002_0016.COM_RxPDO_Map_Outputs_Channel_2.Data_Out[6] <-> COM RxPDO-Map Outputs Channel 2/Data Out 6
//     PlcTask Outputs/GVL_iXlinker.EtherCAT_Master_EPPxxxx.Beckhoff_EPP6xxx.Beckhoff_EPP6xxxEK1122.A_0004_EPP6002_0002_0016.COM_RxPDO_Map_Outputs_Channel_2.Data_Out[7] <-> COM RxPDO-Map Outputs Channel 2/Data Out 7
//     PlcTask Outputs/GVL_iXlinker.EtherCAT_Master_EPPxxxx.Beckhoff_EPP6xxx.Beckhoff_EPP6xxxEK1122.A_0004_EPP6002_0002_0016.COM_RxPDO_Map_Outputs_Channel_2.Data_Out[8] <-> COM RxPDO-Map Outputs Channel 2/Data Out 8
//     PlcTask Outputs/GVL_iXlinker.EtherCAT_Master_EPPxxxx.Beckhoff_EPP6xxx.Beckhoff_EPP6xxxEK1122.A_0004_EPP6002_0002_0016.COM_RxPDO_Map_Outputs_Channel_2.Data_Out[9] <-> COM RxPDO-Map Outputs Channel 2/Data Out 9
//     PlcTask Outputs/GVL_iXlinker.EtherCAT_Master_EPPxxxx.Beckhoff_EPP6xxx.Beckhoff_EPP6xxxEK1122.A_0004_EPP6002_0002_0016.COM_RxPDO_Map_Outputs_Channel_2.Data_Out[10] <-> COM RxPDO-Map Outputs Channel 2/Data Out 10
//     PlcTask Outputs/GVL_iXlinker.EtherCAT_Master_EPPxxxx.Beckhoff_EPP6xxx.Beckhoff_EPP6xxxEK1122.A_0004_EPP6002_0002_0016.COM_RxPDO_Map_Outputs_Channel_2.Data_Out[11] <-> COM RxPDO-Map Outputs Channel 2/Data Out 11
//     PlcTask Outputs/GVL_iXlinker.EtherCAT_Master_EPPxxxx.Beckhoff_EPP6xxx.Beckhoff_EPP6xxxEK1122.A_0004_EPP6002_0002_0016.COM_RxPDO_Map_Outputs_Channel_2.Data_Out[12] <-> COM RxPDO-Map Outputs Channel 2/Data Out 12
//     PlcTask Outputs/GVL_iXlinker.EtherCAT_Master_EPPxxxx.Beckhoff_EPP6xxx.Beckhoff_EPP6xxxEK1122.A_0004_EPP6002_0002_0016.COM_RxPDO_Map_Outputs_Channel_2.Data_Out[13] <-> COM RxPDO-Map Outputs Channel 2/Data Out 13
//     PlcTask Outputs/GVL_iXlinker.EtherCAT_Master_EPPxxxx.Beckhoff_EPP6xxx.Beckhoff_EPP6xxxEK1122.A_0004_EPP6002_0002_0016.COM_RxPDO_Map_Outputs_Channel_2.Data_Out[14] <-> COM RxPDO-Map Outputs Channel 2/Data Out 14
//     PlcTask Outputs/GVL_iXlinker.EtherCAT_Master_EPPxxxx.Beckhoff_EPP6xxx.Beckhoff_EPP6xxxEK1122.A_0004_EPP6002_0002_0016.COM_RxPDO_Map_Outputs_Channel_2.Data_Out[15] <-> COM RxPDO-Map Outputs Channel 2/Data Out 15
//     PlcTask Outputs/GVL_iXlinker.EtherCAT_Master_EPPxxxx.Beckhoff_EPP6xxx.Beckhoff_EPP6xxxEK1122.A_0004_EPP6002_0002_0016.COM_RxPDO_Map_Outputs_Channel_2.Data_Out[16] <-> COM RxPDO-Map Outputs Channel 2/Data Out 16
//     PlcTask Outputs/GVL_iXlinker.EtherCAT_Master_EPPxxxx.Beckhoff_EPP6xxx.Beckhoff_EPP6xxxEK1122.A_0004_EPP6002_0002_0016.COM_RxPDO_Map_Outputs_Channel_2.Data_Out[17] <-> COM RxPDO-Map Outputs Channel 2/Data Out 17
//     PlcTask Outputs/GVL_iXlinker.EtherCAT_Master_EPPxxxx.Beckhoff_EPP6xxx.Beckhoff_EPP6xxxEK1122.A_0004_EPP6002_0002_0016.COM_RxPDO_Map_Outputs_Channel_2.Data_Out[18] <-> COM RxPDO-Map Outputs Channel 2/Data Out 18
//     PlcTask Outputs/GVL_iXlinker.EtherCAT_Master_EPPxxxx.Beckhoff_EPP6xxx.Beckhoff_EPP6xxxEK1122.A_0004_EPP6002_0002_0016.COM_RxPDO_Map_Outputs_Channel_2.Data_Out[19] <-> COM RxPDO-Map Outputs Channel 2/Data Out 19
//     PlcTask Outputs/GVL_iXlinker.EtherCAT_Master_EPPxxxx.Beckhoff_EPP6xxx.Beckhoff_EPP6xxxEK1122.A_0004_EPP6002_0002_0016.COM_RxPDO_Map_Outputs_Channel_2.Data_Out[20] <-> COM RxPDO-Map Outputs Channel 2/Data Out 20
//     PlcTask Outputs/GVL_iXlinker.EtherCAT_Master_EPPxxxx.Beckhoff_EPP6xxx.Beckhoff_EPP6xxxEK1122.A_0004_EPP6002_0002_0016.COM_RxPDO_Map_Outputs_Channel_2.Data_Out[21] <-> COM RxPDO-Map Outputs Channel 2/Data Out 21
//     PlcTask Inputs/GVL_iXlinker.EtherCAT_Master_EPPxxxx.Beckhoff_EPP6xxx.Beckhoff_EPP6xxxEK1122.A_0004_EPP6002_0002_0016.WcState.WcState <-> WcState/WcState
//     PlcTask Inputs/GVL_iXlinker.EtherCAT_Master_EPPxxxx.Beckhoff_EPP6xxx.Beckhoff_EPP6xxxEK1122.A_0004_EPP6002_0002_0016.WcState.InputToggle <-> WcState/InputToggle
//     PlcTask Inputs/GVL_iXlinker.EtherCAT_Master_EPPxxxx.Beckhoff_EPP6xxx.Beckhoff_EPP6xxxEK1122.A_0004_EPP6002_0002_0016.InfoData.AdsAddr <-> InfoData/AdsAddr
//     PlcTask Inputs/GVL_iXlinker.EtherCAT_Master_EPPxxxx.Beckhoff_EPP6xxx.Beckhoff_EPP6xxxEK1122.A_0004_EPP6002_0002_0016.InfoData.State <-> InfoData/State
//   PLC/PLC Instance <-> EtherCAT Master EPPxxxx/Beckhoff EPP6xxx/Beckhoff EPP6xxxEK1122/A_0005(EPP6002-0002-0017)
//     PlcTask Inputs/GVL_iXlinker.EtherCAT_Master_EPPxxxx.Beckhoff_EPP6xxx.Beckhoff_EPP6xxxEK1122.A_0005_EPP6002_0002_0017.COM_TxPDO_Map_Inputs_Channel_1.Status <-> COM TxPDO-Map Inputs Channel 1/Status
//     PlcTask Inputs/GVL_iXlinker.EtherCAT_Master_EPPxxxx.Beckhoff_EPP6xxx.Beckhoff_EPP6xxxEK1122.A_0005_EPP6002_0002_0017.COM_TxPDO_Map_Inputs_Channel_2.Status <-> COM TxPDO-Map Inputs Channel 2/Status
//     PlcTask Inputs/GVL_iXlinker.EtherCAT_Master_EPPxxxx.Beckhoff_EPP6xxx.Beckhoff_EPP6xxxEK1122.A_0005_EPP6002_0002_0017.COM_TxPDO_Map_Inputs_Channel_1.Data_In[0] <-> COM TxPDO-Map Inputs Channel 1/Data In 0
//     PlcTask Inputs/GVL_iXlinker.EtherCAT_Master_EPPxxxx.Beckhoff_EPP6xxx.Beckhoff_EPP6xxxEK1122.A_0005_EPP6002_0002_0017.COM_TxPDO_Map_Inputs_Channel_1.Data_In[1] <-> COM TxPDO-Map Inputs Channel 1/Data In 1
//     PlcTask Inputs/GVL_iXlinker.EtherCAT_Master_EPPxxxx.Beckhoff_EPP6xxx.Beckhoff_EPP6xxxEK1122.A_0005_EPP6002_0002_0017.COM_TxPDO_Map_Inputs_Channel_1.Data_In[2] <-> COM TxPDO-Map Inputs Channel 1/Data In 2
//     PlcTask Inputs/GVL_iXlinker.EtherCAT_Master_EPPxxxx.Beckhoff_EPP6xxx.Beckhoff_EPP6xxxEK1122.A_0005_EPP6002_0002_0017.COM_TxPDO_Map_Inputs_Channel_1.Data_In[3] <-> COM TxPDO-Map Inputs Channel 1/Data In 3
//     PlcTask Inputs/GVL_iXlinker.EtherCAT_Master_EPPxxxx.Beckhoff_EPP6xxx.Beckhoff_EPP6xxxEK1122.A_0005_EPP6002_0002_0017.COM_TxPDO_Map_Inputs_Channel_1.Data_In[4] <-> COM TxPDO-Map Inputs Channel 1/Data In 4
//     PlcTask Inputs/GVL_iXlinker.EtherCAT_Master_EPPxxxx.Beckhoff_EPP6xxx.Beckhoff_EPP6xxxEK1122.A_0005_EPP6002_0002_0017.COM_TxPDO_Map_Inputs_Channel_1.Data_In[5] <-> COM TxPDO-Map Inputs Channel 1/Data In 5
//     PlcTask Inputs/GVL_iXlinker.EtherCAT_Master_EPPxxxx.Beckhoff_EPP6xxx.Beckhoff_EPP6xxxEK1122.A_0005_EPP6002_0002_0017.COM_TxPDO_Map_Inputs_Channel_1.Data_In[6] <-> COM TxPDO-Map Inputs Channel 1/Data In 6
//     PlcTask Inputs/GVL_iXlinker.EtherCAT_Master_EPPxxxx.Beckhoff_EPP6xxx.Beckhoff_EPP6xxxEK1122.A_0005_EPP6002_0002_0017.COM_TxPDO_Map_Inputs_Channel_1.Data_In[7] <-> COM TxPDO-Map Inputs Channel 1/Data In 7
//     PlcTask Inputs/GVL_iXlinker.EtherCAT_Master_EPPxxxx.Beckhoff_EPP6xxx.Beckhoff_EPP6xxxEK1122.A_0005_EPP6002_0002_0017.COM_TxPDO_Map_Inputs_Channel_1.Data_In[8] <-> COM TxPDO-Map Inputs Channel 1/Data In 8
//     PlcTask Inputs/GVL_iXlinker.EtherCAT_Master_EPPxxxx.Beckhoff_EPP6xxx.Beckhoff_EPP6xxxEK1122.A_0005_EPP6002_0002_0017.COM_TxPDO_Map_Inputs_Channel_1.Data_In[9] <-> COM TxPDO-Map Inputs Channel 1/Data In 9
//     PlcTask Inputs/GVL_iXlinker.EtherCAT_Master_EPPxxxx.Beckhoff_EPP6xxx.Beckhoff_EPP6xxxEK1122.A_0005_EPP6002_0002_0017.COM_TxPDO_Map_Inputs_Channel_1.Data_In[10] <-> COM TxPDO-Map Inputs Channel 1/Data In 10
//     PlcTask Inputs/GVL_iXlinker.EtherCAT_Master_EPPxxxx.Beckhoff_EPP6xxx.Beckhoff_EPP6xxxEK1122.A_0005_EPP6002_0002_0017.COM_TxPDO_Map_Inputs_Channel_1.Data_In[11] <-> COM TxPDO-Map Inputs Channel 1/Data In 11
//     PlcTask Inputs/GVL_iXlinker.EtherCAT_Master_EPPxxxx.Beckhoff_EPP6xxx.Beckhoff_EPP6xxxEK1122.A_0005_EPP6002_0002_0017.COM_TxPDO_Map_Inputs_Channel_1.Data_In[12] <-> COM TxPDO-Map Inputs Channel 1/Data In 12
//     PlcTask Inputs/GVL_iXlinker.EtherCAT_Master_EPPxxxx.Beckhoff_EPP6xxx.Beckhoff_EPP6xxxEK1122.A_0005_EPP6002_0002_0017.COM_TxPDO_Map_Inputs_Channel_1.Data_In[13] <-> COM TxPDO-Map Inputs Channel 1/Data In 13
//     PlcTask Inputs/GVL_iXlinker.EtherCAT_Master_EPPxxxx.Beckhoff_EPP6xxx.Beckhoff_EPP6xxxEK1122.A_0005_EPP6002_0002_0017.COM_TxPDO_Map_Inputs_Channel_1.Data_In[14] <-> COM TxPDO-Map Inputs Channel 1/Data In 14
//     PlcTask Inputs/GVL_iXlinker.EtherCAT_Master_EPPxxxx.Beckhoff_EPP6xxx.Beckhoff_EPP6xxxEK1122.A_0005_EPP6002_0002_0017.COM_TxPDO_Map_Inputs_Channel_1.Data_In[15] <-> COM TxPDO-Map Inputs Channel 1/Data In 15
//     PlcTask Inputs/GVL_iXlinker.EtherCAT_Master_EPPxxxx.Beckhoff_EPP6xxx.Beckhoff_EPP6xxxEK1122.A_0005_EPP6002_0002_0017.COM_TxPDO_Map_Inputs_Channel_1.Data_In[16] <-> COM TxPDO-Map Inputs Channel 1/Data In 16
//     PlcTask Inputs/GVL_iXlinker.EtherCAT_Master_EPPxxxx.Beckhoff_EPP6xxx.Beckhoff_EPP6xxxEK1122.A_0005_EPP6002_0002_0017.COM_TxPDO_Map_Inputs_Channel_1.Data_In[17] <-> COM TxPDO-Map Inputs Channel 1/Data In 17
//     PlcTask Inputs/GVL_iXlinker.EtherCAT_Master_EPPxxxx.Beckhoff_EPP6xxx.Beckhoff_EPP6xxxEK1122.A_0005_EPP6002_0002_0017.COM_TxPDO_Map_Inputs_Channel_1.Data_In[18] <-> COM TxPDO-Map Inputs Channel 1/Data In 18
//     PlcTask Inputs/GVL_iXlinker.EtherCAT_Master_EPPxxxx.Beckhoff_EPP6xxx.Beckhoff_EPP6xxxEK1122.A_0005_EPP6002_0002_0017.COM_TxPDO_Map_Inputs_Channel_1.Data_In[19] <-> COM TxPDO-Map Inputs Channel 1/Data In 19
//     PlcTask Inputs/GVL_iXlinker.EtherCAT_Master_EPPxxxx.Beckhoff_EPP6xxx.Beckhoff_EPP6xxxEK1122.A_0005_EPP6002_0002_0017.COM_TxPDO_Map_Inputs_Channel_1.Data_In[20] <-> COM TxPDO-Map Inputs Channel 1/Data In 20
//     PlcTask Inputs/GVL_iXlinker.EtherCAT_Master_EPPxxxx.Beckhoff_EPP6xxx.Beckhoff_EPP6xxxEK1122.A_0005_EPP6002_0002_0017.COM_TxPDO_Map_Inputs_Channel_1.Data_In[21] <-> COM TxPDO-Map Inputs Channel 1/Data In 21
//     PlcTask Inputs/GVL_iXlinker.EtherCAT_Master_EPPxxxx.Beckhoff_EPP6xxx.Beckhoff_EPP6xxxEK1122.A_0005_EPP6002_0002_0017.COM_TxPDO_Map_Inputs_Channel_2.Data_In[0] <-> COM TxPDO-Map Inputs Channel 2/Data In 0
//     PlcTask Inputs/GVL_iXlinker.EtherCAT_Master_EPPxxxx.Beckhoff_EPP6xxx.Beckhoff_EPP6xxxEK1122.A_0005_EPP6002_0002_0017.COM_TxPDO_Map_Inputs_Channel_2.Data_In[1] <-> COM TxPDO-Map Inputs Channel 2/Data In 1
//     PlcTask Inputs/GVL_iXlinker.EtherCAT_Master_EPPxxxx.Beckhoff_EPP6xxx.Beckhoff_EPP6xxxEK1122.A_0005_EPP6002_0002_0017.COM_TxPDO_Map_Inputs_Channel_2.Data_In[2] <-> COM TxPDO-Map Inputs Channel 2/Data In 2
//     PlcTask Inputs/GVL_iXlinker.EtherCAT_Master_EPPxxxx.Beckhoff_EPP6xxx.Beckhoff_EPP6xxxEK1122.A_0005_EPP6002_0002_0017.COM_TxPDO_Map_Inputs_Channel_2.Data_In[3] <-> COM TxPDO-Map Inputs Channel 2/Data In 3
//     PlcTask Inputs/GVL_iXlinker.EtherCAT_Master_EPPxxxx.Beckhoff_EPP6xxx.Beckhoff_EPP6xxxEK1122.A_0005_EPP6002_0002_0017.COM_TxPDO_Map_Inputs_Channel_2.Data_In[4] <-> COM TxPDO-Map Inputs Channel 2/Data In 4
//     PlcTask Inputs/GVL_iXlinker.EtherCAT_Master_EPPxxxx.Beckhoff_EPP6xxx.Beckhoff_EPP6xxxEK1122.A_0005_EPP6002_0002_0017.COM_TxPDO_Map_Inputs_Channel_2.Data_In[5] <-> COM TxPDO-Map Inputs Channel 2/Data In 5
//     PlcTask Inputs/GVL_iXlinker.EtherCAT_Master_EPPxxxx.Beckhoff_EPP6xxx.Beckhoff_EPP6xxxEK1122.A_0005_EPP6002_0002_0017.COM_TxPDO_Map_Inputs_Channel_2.Data_In[6] <-> COM TxPDO-Map Inputs Channel 2/Data In 6
//     PlcTask Inputs/GVL_iXlinker.EtherCAT_Master_EPPxxxx.Beckhoff_EPP6xxx.Beckhoff_EPP6xxxEK1122.A_0005_EPP6002_0002_0017.COM_TxPDO_Map_Inputs_Channel_2.Data_In[7] <-> COM TxPDO-Map Inputs Channel 2/Data In 7
//     PlcTask Inputs/GVL_iXlinker.EtherCAT_Master_EPPxxxx.Beckhoff_EPP6xxx.Beckhoff_EPP6xxxEK1122.A_0005_EPP6002_0002_0017.COM_TxPDO_Map_Inputs_Channel_2.Data_In[8] <-> COM TxPDO-Map Inputs Channel 2/Data In 8
//     PlcTask Inputs/GVL_iXlinker.EtherCAT_Master_EPPxxxx.Beckhoff_EPP6xxx.Beckhoff_EPP6xxxEK1122.A_0005_EPP6002_0002_0017.COM_TxPDO_Map_Inputs_Channel_2.Data_In[9] <-> COM TxPDO-Map Inputs Channel 2/Data In 9
//     PlcTask Inputs/GVL_iXlinker.EtherCAT_Master_EPPxxxx.Beckhoff_EPP6xxx.Beckhoff_EPP6xxxEK1122.A_0005_EPP6002_0002_0017.COM_TxPDO_Map_Inputs_Channel_2.Data_In[10] <-> COM TxPDO-Map Inputs Channel 2/Data In 10
//     PlcTask Inputs/GVL_iXlinker.EtherCAT_Master_EPPxxxx.Beckhoff_EPP6xxx.Beckhoff_EPP6xxxEK1122.A_0005_EPP6002_0002_0017.COM_TxPDO_Map_Inputs_Channel_2.Data_In[11] <-> COM TxPDO-Map Inputs Channel 2/Data In 11
//     PlcTask Inputs/GVL_iXlinker.EtherCAT_Master_EPPxxxx.Beckhoff_EPP6xxx.Beckhoff_EPP6xxxEK1122.A_0005_EPP6002_0002_0017.COM_TxPDO_Map_Inputs_Channel_2.Data_In[12] <-> COM TxPDO-Map Inputs Channel 2/Data In 12
//     PlcTask Inputs/GVL_iXlinker.EtherCAT_Master_EPPxxxx.Beckhoff_EPP6xxx.Beckhoff_EPP6xxxEK1122.A_0005_EPP6002_0002_0017.COM_TxPDO_Map_Inputs_Channel_2.Data_In[13] <-> COM TxPDO-Map Inputs Channel 2/Data In 13
//     PlcTask Inputs/GVL_iXlinker.EtherCAT_Master_EPPxxxx.Beckhoff_EPP6xxx.Beckhoff_EPP6xxxEK1122.A_0005_EPP6002_0002_0017.COM_TxPDO_Map_Inputs_Channel_2.Data_In[14] <-> COM TxPDO-Map Inputs Channel 2/Data In 14
//     PlcTask Inputs/GVL_iXlinker.EtherCAT_Master_EPPxxxx.Beckhoff_EPP6xxx.Beckhoff_EPP6xxxEK1122.A_0005_EPP6002_0002_0017.COM_TxPDO_Map_Inputs_Channel_2.Data_In[15] <-> COM TxPDO-Map Inputs Channel 2/Data In 15
//     PlcTask Inputs/GVL_iXlinker.EtherCAT_Master_EPPxxxx.Beckhoff_EPP6xxx.Beckhoff_EPP6xxxEK1122.A_0005_EPP6002_0002_0017.COM_TxPDO_Map_Inputs_Channel_2.Data_In[16] <-> COM TxPDO-Map Inputs Channel 2/Data In 16
//     PlcTask Inputs/GVL_iXlinker.EtherCAT_Master_EPPxxxx.Beckhoff_EPP6xxx.Beckhoff_EPP6xxxEK1122.A_0005_EPP6002_0002_0017.COM_TxPDO_Map_Inputs_Channel_2.Data_In[17] <-> COM TxPDO-Map Inputs Channel 2/Data In 17
//     PlcTask Inputs/GVL_iXlinker.EtherCAT_Master_EPPxxxx.Beckhoff_EPP6xxx.Beckhoff_EPP6xxxEK1122.A_0005_EPP6002_0002_0017.COM_TxPDO_Map_Inputs_Channel_2.Data_In[18] <-> COM TxPDO-Map Inputs Channel 2/Data In 18
//     PlcTask Inputs/GVL_iXlinker.EtherCAT_Master_EPPxxxx.Beckhoff_EPP6xxx.Beckhoff_EPP6xxxEK1122.A_0005_EPP6002_0002_0017.COM_TxPDO_Map_Inputs_Channel_2.Data_In[19] <-> COM TxPDO-Map Inputs Channel 2/Data In 19
//     PlcTask Inputs/GVL_iXlinker.EtherCAT_Master_EPPxxxx.Beckhoff_EPP6xxx.Beckhoff_EPP6xxxEK1122.A_0005_EPP6002_0002_0017.COM_TxPDO_Map_Inputs_Channel_2.Data_In[20] <-> COM TxPDO-Map Inputs Channel 2/Data In 20
//     PlcTask Inputs/GVL_iXlinker.EtherCAT_Master_EPPxxxx.Beckhoff_EPP6xxx.Beckhoff_EPP6xxxEK1122.A_0005_EPP6002_0002_0017.COM_TxPDO_Map_Inputs_Channel_2.Data_In[21] <-> COM TxPDO-Map Inputs Channel 2/Data In 21
//     PlcTask Outputs/GVL_iXlinker.EtherCAT_Master_EPPxxxx.Beckhoff_EPP6xxx.Beckhoff_EPP6xxxEK1122.A_0005_EPP6002_0002_0017.COM_RxPDO_Map_Outputs_Channel_1.Ctrl <-> COM RxPDO-Map Outputs Channel 1/Ctrl
//     PlcTask Outputs/GVL_iXlinker.EtherCAT_Master_EPPxxxx.Beckhoff_EPP6xxx.Beckhoff_EPP6xxxEK1122.A_0005_EPP6002_0002_0017.COM_RxPDO_Map_Outputs_Channel_2.Ctrl <-> COM RxPDO-Map Outputs Channel 2/Ctrl
//     PlcTask Outputs/GVL_iXlinker.EtherCAT_Master_EPPxxxx.Beckhoff_EPP6xxx.Beckhoff_EPP6xxxEK1122.A_0005_EPP6002_0002_0017.COM_RxPDO_Map_Outputs_Channel_1.Data_Out[0] <-> COM RxPDO-Map Outputs Channel 1/Data Out 0
//     PlcTask Outputs/GVL_iXlinker.EtherCAT_Master_EPPxxxx.Beckhoff_EPP6xxx.Beckhoff_EPP6xxxEK1122.A_0005_EPP6002_0002_0017.COM_RxPDO_Map_Outputs_Channel_1.Data_Out[1] <-> COM RxPDO-Map Outputs Channel 1/Data Out 1
//     PlcTask Outputs/GVL_iXlinker.EtherCAT_Master_EPPxxxx.Beckhoff_EPP6xxx.Beckhoff_EPP6xxxEK1122.A_0005_EPP6002_0002_0017.COM_RxPDO_Map_Outputs_Channel_1.Data_Out[2] <-> COM RxPDO-Map Outputs Channel 1/Data Out 2
//     PlcTask Outputs/GVL_iXlinker.EtherCAT_Master_EPPxxxx.Beckhoff_EPP6xxx.Beckhoff_EPP6xxxEK1122.A_0005_EPP6002_0002_0017.COM_RxPDO_Map_Outputs_Channel_1.Data_Out[3] <-> COM RxPDO-Map Outputs Channel 1/Data Out 3
//     PlcTask Outputs/GVL_iXlinker.EtherCAT_Master_EPPxxxx.Beckhoff_EPP6xxx.Beckhoff_EPP6xxxEK1122.A_0005_EPP6002_0002_0017.COM_RxPDO_Map_Outputs_Channel_1.Data_Out[4] <-> COM RxPDO-Map Outputs Channel 1/Data Out 4
//     PlcTask Outputs/GVL_iXlinker.EtherCAT_Master_EPPxxxx.Beckhoff_EPP6xxx.Beckhoff_EPP6xxxEK1122.A_0005_EPP6002_0002_0017.COM_RxPDO_Map_Outputs_Channel_1.Data_Out[5] <-> COM RxPDO-Map Outputs Channel 1/Data Out 5
//     PlcTask Outputs/GVL_iXlinker.EtherCAT_Master_EPPxxxx.Beckhoff_EPP6xxx.Beckhoff_EPP6xxxEK1122.A_0005_EPP6002_0002_0017.COM_RxPDO_Map_Outputs_Channel_1.Data_Out[6] <-> COM RxPDO-Map Outputs Channel 1/Data Out 6
//     PlcTask Outputs/GVL_iXlinker.EtherCAT_Master_EPPxxxx.Beckhoff_EPP6xxx.Beckhoff_EPP6xxxEK1122.A_0005_EPP6002_0002_0017.COM_RxPDO_Map_Outputs_Channel_1.Data_Out[7] <-> COM RxPDO-Map Outputs Channel 1/Data Out 7
//     PlcTask Outputs/GVL_iXlinker.EtherCAT_Master_EPPxxxx.Beckhoff_EPP6xxx.Beckhoff_EPP6xxxEK1122.A_0005_EPP6002_0002_0017.COM_RxPDO_Map_Outputs_Channel_1.Data_Out[8] <-> COM RxPDO-Map Outputs Channel 1/Data Out 8
//     PlcTask Outputs/GVL_iXlinker.EtherCAT_Master_EPPxxxx.Beckhoff_EPP6xxx.Beckhoff_EPP6xxxEK1122.A_0005_EPP6002_0002_0017.COM_RxPDO_Map_Outputs_Channel_1.Data_Out[9] <-> COM RxPDO-Map Outputs Channel 1/Data Out 9
//     PlcTask Outputs/GVL_iXlinker.EtherCAT_Master_EPPxxxx.Beckhoff_EPP6xxx.Beckhoff_EPP6xxxEK1122.A_0005_EPP6002_0002_0017.COM_RxPDO_Map_Outputs_Channel_1.Data_Out[10] <-> COM RxPDO-Map Outputs Channel 1/Data Out 10
//     PlcTask Outputs/GVL_iXlinker.EtherCAT_Master_EPPxxxx.Beckhoff_EPP6xxx.Beckhoff_EPP6xxxEK1122.A_0005_EPP6002_0002_0017.COM_RxPDO_Map_Outputs_Channel_1.Data_Out[11] <-> COM RxPDO-Map Outputs Channel 1/Data Out 11
//     PlcTask Outputs/GVL_iXlinker.EtherCAT_Master_EPPxxxx.Beckhoff_EPP6xxx.Beckhoff_EPP6xxxEK1122.A_0005_EPP6002_0002_0017.COM_RxPDO_Map_Outputs_Channel_1.Data_Out[12] <-> COM RxPDO-Map Outputs Channel 1/Data Out 12
//     PlcTask Outputs/GVL_iXlinker.EtherCAT_Master_EPPxxxx.Beckhoff_EPP6xxx.Beckhoff_EPP6xxxEK1122.A_0005_EPP6002_0002_0017.COM_RxPDO_Map_Outputs_Channel_1.Data_Out[13] <-> COM RxPDO-Map Outputs Channel 1/Data Out 13
//     PlcTask Outputs/GVL_iXlinker.EtherCAT_Master_EPPxxxx.Beckhoff_EPP6xxx.Beckhoff_EPP6xxxEK1122.A_0005_EPP6002_0002_0017.COM_RxPDO_Map_Outputs_Channel_1.Data_Out[14] <-> COM RxPDO-Map Outputs Channel 1/Data Out 14
//     PlcTask Outputs/GVL_iXlinker.EtherCAT_Master_EPPxxxx.Beckhoff_EPP6xxx.Beckhoff_EPP6xxxEK1122.A_0005_EPP6002_0002_0017.COM_RxPDO_Map_Outputs_Channel_1.Data_Out[15] <-> COM RxPDO-Map Outputs Channel 1/Data Out 15
//     PlcTask Outputs/GVL_iXlinker.EtherCAT_Master_EPPxxxx.Beckhoff_EPP6xxx.Beckhoff_EPP6xxxEK1122.A_0005_EPP6002_0002_0017.COM_RxPDO_Map_Outputs_Channel_1.Data_Out[16] <-> COM RxPDO-Map Outputs Channel 1/Data Out 16
//     PlcTask Outputs/GVL_iXlinker.EtherCAT_Master_EPPxxxx.Beckhoff_EPP6xxx.Beckhoff_EPP6xxxEK1122.A_0005_EPP6002_0002_0017.COM_RxPDO_Map_Outputs_Channel_1.Data_Out[17] <-> COM RxPDO-Map Outputs Channel 1/Data Out 17
//     PlcTask Outputs/GVL_iXlinker.EtherCAT_Master_EPPxxxx.Beckhoff_EPP6xxx.Beckhoff_EPP6xxxEK1122.A_0005_EPP6002_0002_0017.COM_RxPDO_Map_Outputs_Channel_1.Data_Out[18] <-> COM RxPDO-Map Outputs Channel 1/Data Out 18
//     PlcTask Outputs/GVL_iXlinker.EtherCAT_Master_EPPxxxx.Beckhoff_EPP6xxx.Beckhoff_EPP6xxxEK1122.A_0005_EPP6002_0002_0017.COM_RxPDO_Map_Outputs_Channel_1.Data_Out[19] <-> COM RxPDO-Map Outputs Channel 1/Data Out 19
//     PlcTask Outputs/GVL_iXlinker.EtherCAT_Master_EPPxxxx.Beckhoff_EPP6xxx.Beckhoff_EPP6xxxEK1122.A_0005_EPP6002_0002_0017.COM_RxPDO_Map_Outputs_Channel_1.Data_Out[20] <-> COM RxPDO-Map Outputs Channel 1/Data Out 20
//     PlcTask Outputs/GVL_iXlinker.EtherCAT_Master_EPPxxxx.Beckhoff_EPP6xxx.Beckhoff_EPP6xxxEK1122.A_0005_EPP6002_0002_0017.COM_RxPDO_Map_Outputs_Channel_1.Data_Out[21] <-> COM RxPDO-Map Outputs Channel 1/Data Out 21
//     PlcTask Outputs/GVL_iXlinker.EtherCAT_Master_EPPxxxx.Beckhoff_EPP6xxx.Beckhoff_EPP6xxxEK1122.A_0005_EPP6002_0002_0017.COM_RxPDO_Map_Outputs_Channel_2.Data_Out[0] <-> COM RxPDO-Map Outputs Channel 2/Data Out 0
//     PlcTask Outputs/GVL_iXlinker.EtherCAT_Master_EPPxxxx.Beckhoff_EPP6xxx.Beckhoff_EPP6xxxEK1122.A_0005_EPP6002_0002_0017.COM_RxPDO_Map_Outputs_Channel_2.Data_Out[1] <-> COM RxPDO-Map Outputs Channel 2/Data Out 1
//     PlcTask Outputs/GVL_iXlinker.EtherCAT_Master_EPPxxxx.Beckhoff_EPP6xxx.Beckhoff_EPP6xxxEK1122.A_0005_EPP6002_0002_0017.COM_RxPDO_Map_Outputs_Channel_2.Data_Out[2] <-> COM RxPDO-Map Outputs Channel 2/Data Out 2
//     PlcTask Outputs/GVL_iXlinker.EtherCAT_Master_EPPxxxx.Beckhoff_EPP6xxx.Beckhoff_EPP6xxxEK1122.A_0005_EPP6002_0002_0017.COM_RxPDO_Map_Outputs_Channel_2.Data_Out[3] <-> COM RxPDO-Map Outputs Channel 2/Data Out 3
//     PlcTask Outputs/GVL_iXlinker.EtherCAT_Master_EPPxxxx.Beckhoff_EPP6xxx.Beckhoff_EPP6xxxEK1122.A_0005_EPP6002_0002_0017.COM_RxPDO_Map_Outputs_Channel_2.Data_Out[4] <-> COM RxPDO-Map Outputs Channel 2/Data Out 4
//     PlcTask Outputs/GVL_iXlinker.EtherCAT_Master_EPPxxxx.Beckhoff_EPP6xxx.Beckhoff_EPP6xxxEK1122.A_0005_EPP6002_0002_0017.COM_RxPDO_Map_Outputs_Channel_2.Data_Out[5] <-> COM RxPDO-Map Outputs Channel 2/Data Out 5
//     PlcTask Outputs/GVL_iXlinker.EtherCAT_Master_EPPxxxx.Beckhoff_EPP6xxx.Beckhoff_EPP6xxxEK1122.A_0005_EPP6002_0002_0017.COM_RxPDO_Map_Outputs_Channel_2.Data_Out[6] <-> COM RxPDO-Map Outputs Channel 2/Data Out 6
//     PlcTask Outputs/GVL_iXlinker.EtherCAT_Master_EPPxxxx.Beckhoff_EPP6xxx.Beckhoff_EPP6xxxEK1122.A_0005_EPP6002_0002_0017.COM_RxPDO_Map_Outputs_Channel_2.Data_Out[7] <-> COM RxPDO-Map Outputs Channel 2/Data Out 7
//     PlcTask Outputs/GVL_iXlinker.EtherCAT_Master_EPPxxxx.Beckhoff_EPP6xxx.Beckhoff_EPP6xxxEK1122.A_0005_EPP6002_0002_0017.COM_RxPDO_Map_Outputs_Channel_2.Data_Out[8] <-> COM RxPDO-Map Outputs Channel 2/Data Out 8
//     PlcTask Outputs/GVL_iXlinker.EtherCAT_Master_EPPxxxx.Beckhoff_EPP6xxx.Beckhoff_EPP6xxxEK1122.A_0005_EPP6002_0002_0017.COM_RxPDO_Map_Outputs_Channel_2.Data_Out[9] <-> COM RxPDO-Map Outputs Channel 2/Data Out 9
//     PlcTask Outputs/GVL_iXlinker.EtherCAT_Master_EPPxxxx.Beckhoff_EPP6xxx.Beckhoff_EPP6xxxEK1122.A_0005_EPP6002_0002_0017.COM_RxPDO_Map_Outputs_Channel_2.Data_Out[10] <-> COM RxPDO-Map Outputs Channel 2/Data Out 10
//     PlcTask Outputs/GVL_iXlinker.EtherCAT_Master_EPPxxxx.Beckhoff_EPP6xxx.Beckhoff_EPP6xxxEK1122.A_0005_EPP6002_0002_0017.COM_RxPDO_Map_Outputs_Channel_2.Data_Out[11] <-> COM RxPDO-Map Outputs Channel 2/Data Out 11
//     PlcTask Outputs/GVL_iXlinker.EtherCAT_Master_EPPxxxx.Beckhoff_EPP6xxx.Beckhoff_EPP6xxxEK1122.A_0005_EPP6002_0002_0017.COM_RxPDO_Map_Outputs_Channel_2.Data_Out[12] <-> COM RxPDO-Map Outputs Channel 2/Data Out 12
//     PlcTask Outputs/GVL_iXlinker.EtherCAT_Master_EPPxxxx.Beckhoff_EPP6xxx.Beckhoff_EPP6xxxEK1122.A_0005_EPP6002_0002_0017.COM_RxPDO_Map_Outputs_Channel_2.Data_Out[13] <-> COM RxPDO-Map Outputs Channel 2/Data Out 13
//     PlcTask Outputs/GVL_iXlinker.EtherCAT_Master_EPPxxxx.Beckhoff_EPP6xxx.Beckhoff_EPP6xxxEK1122.A_0005_EPP6002_0002_0017.COM_RxPDO_Map_Outputs_Channel_2.Data_Out[14] <-> COM RxPDO-Map Outputs Channel 2/Data Out 14
//     PlcTask Outputs/GVL_iXlinker.EtherCAT_Master_EPPxxxx.Beckhoff_EPP6xxx.Beckhoff_EPP6xxxEK1122.A_0005_EPP6002_0002_0017.COM_RxPDO_Map_Outputs_Channel_2.Data_Out[15] <-> COM RxPDO-Map Outputs Channel 2/Data Out 15
//     PlcTask Outputs/GVL_iXlinker.EtherCAT_Master_EPPxxxx.Beckhoff_EPP6xxx.Beckhoff_EPP6xxxEK1122.A_0005_EPP6002_0002_0017.COM_RxPDO_Map_Outputs_Channel_2.Data_Out[16] <-> COM RxPDO-Map Outputs Channel 2/Data Out 16
//     PlcTask Outputs/GVL_iXlinker.EtherCAT_Master_EPPxxxx.Beckhoff_EPP6xxx.Beckhoff_EPP6xxxEK1122.A_0005_EPP6002_0002_0017.COM_RxPDO_Map_Outputs_Channel_2.Data_Out[17] <-> COM RxPDO-Map Outputs Channel 2/Data Out 17
//     PlcTask Outputs/GVL_iXlinker.EtherCAT_Master_EPPxxxx.Beckhoff_EPP6xxx.Beckhoff_EPP6xxxEK1122.A_0005_EPP6002_0002_0017.COM_RxPDO_Map_Outputs_Channel_2.Data_Out[18] <-> COM RxPDO-Map Outputs Channel 2/Data Out 18
//     PlcTask Outputs/GVL_iXlinker.EtherCAT_Master_EPPxxxx.Beckhoff_EPP6xxx.Beckhoff_EPP6xxxEK1122.A_0005_EPP6002_0002_0017.COM_RxPDO_Map_Outputs_Channel_2.Data_Out[19] <-> COM RxPDO-Map Outputs Channel 2/Data Out 19
//     PlcTask Outputs/GVL_iXlinker.EtherCAT_Master_EPPxxxx.Beckhoff_EPP6xxx.Beckhoff_EPP6xxxEK1122.A_0005_EPP6002_0002_0017.COM_RxPDO_Map_Outputs_Channel_2.Data_Out[20] <-> COM RxPDO-Map Outputs Channel 2/Data Out 20
//     PlcTask Outputs/GVL_iXlinker.EtherCAT_Master_EPPxxxx.Beckhoff_EPP6xxx.Beckhoff_EPP6xxxEK1122.A_0005_EPP6002_0002_0017.COM_RxPDO_Map_Outputs_Channel_2.Data_Out[21] <-> COM RxPDO-Map Outputs Channel 2/Data Out 21
//     PlcTask Inputs/GVL_iXlinker.EtherCAT_Master_EPPxxxx.Beckhoff_EPP6xxx.Beckhoff_EPP6xxxEK1122.A_0005_EPP6002_0002_0017.WcState.WcState <-> WcState/WcState
//     PlcTask Inputs/GVL_iXlinker.EtherCAT_Master_EPPxxxx.Beckhoff_EPP6xxx.Beckhoff_EPP6xxxEK1122.A_0005_EPP6002_0002_0017.WcState.InputToggle <-> WcState/InputToggle
//     PlcTask Inputs/GVL_iXlinker.EtherCAT_Master_EPPxxxx.Beckhoff_EPP6xxx.Beckhoff_EPP6xxxEK1122.A_0005_EPP6002_0002_0017.InfoData.AdsAddr <-> InfoData/AdsAddr
//     PlcTask Inputs/GVL_iXlinker.EtherCAT_Master_EPPxxxx.Beckhoff_EPP6xxx.Beckhoff_EPP6xxxEK1122.A_0005_EPP6002_0002_0017.InfoData.State <-> InfoData/State
//   PLC/PLC Instance <-> EtherCAT Master EPPxxxx/Beckhoff EPP6xxx/Beckhoff EPP6xxxEK1122/A_0006(EPP6002-0002-0018)
//     PlcTask Inputs/GVL_iXlinker.EtherCAT_Master_EPPxxxx.Beckhoff_EPP6xxx.Beckhoff_EPP6xxxEK1122.A_0006_EPP6002_0002_0018.COM_TxPDO_Map_Inputs_Channel_1.Status <-> COM TxPDO-Map Inputs Channel 1/Status
//     PlcTask Inputs/GVL_iXlinker.EtherCAT_Master_EPPxxxx.Beckhoff_EPP6xxx.Beckhoff_EPP6xxxEK1122.A_0006_EPP6002_0002_0018.COM_TxPDO_Map_Inputs_Channel_2.Status <-> COM TxPDO-Map Inputs Channel 2/Status
//     PlcTask Inputs/GVL_iXlinker.EtherCAT_Master_EPPxxxx.Beckhoff_EPP6xxx.Beckhoff_EPP6xxxEK1122.A_0006_EPP6002_0002_0018.COM_TxPDO_Map_Inputs_Channel_1.Data_In[0] <-> COM TxPDO-Map Inputs Channel 1/Data In 0
//     PlcTask Inputs/GVL_iXlinker.EtherCAT_Master_EPPxxxx.Beckhoff_EPP6xxx.Beckhoff_EPP6xxxEK1122.A_0006_EPP6002_0002_0018.COM_TxPDO_Map_Inputs_Channel_1.Data_In[1] <-> COM TxPDO-Map Inputs Channel 1/Data In 1
//     PlcTask Inputs/GVL_iXlinker.EtherCAT_Master_EPPxxxx.Beckhoff_EPP6xxx.Beckhoff_EPP6xxxEK1122.A_0006_EPP6002_0002_0018.COM_TxPDO_Map_Inputs_Channel_1.Data_In[2] <-> COM TxPDO-Map Inputs Channel 1/Data In 2
//     PlcTask Inputs/GVL_iXlinker.EtherCAT_Master_EPPxxxx.Beckhoff_EPP6xxx.Beckhoff_EPP6xxxEK1122.A_0006_EPP6002_0002_0018.COM_TxPDO_Map_Inputs_Channel_1.Data_In[3] <-> COM TxPDO-Map Inputs Channel 1/Data In 3
//     PlcTask Inputs/GVL_iXlinker.EtherCAT_Master_EPPxxxx.Beckhoff_EPP6xxx.Beckhoff_EPP6xxxEK1122.A_0006_EPP6002_0002_0018.COM_TxPDO_Map_Inputs_Channel_1.Data_In[4] <-> COM TxPDO-Map Inputs Channel 1/Data In 4
//     PlcTask Inputs/GVL_iXlinker.EtherCAT_Master_EPPxxxx.Beckhoff_EPP6xxx.Beckhoff_EPP6xxxEK1122.A_0006_EPP6002_0002_0018.COM_TxPDO_Map_Inputs_Channel_1.Data_In[5] <-> COM TxPDO-Map Inputs Channel 1/Data In 5
//     PlcTask Inputs/GVL_iXlinker.EtherCAT_Master_EPPxxxx.Beckhoff_EPP6xxx.Beckhoff_EPP6xxxEK1122.A_0006_EPP6002_0002_0018.COM_TxPDO_Map_Inputs_Channel_1.Data_In[6] <-> COM TxPDO-Map Inputs Channel 1/Data In 6
//     PlcTask Inputs/GVL_iXlinker.EtherCAT_Master_EPPxxxx.Beckhoff_EPP6xxx.Beckhoff_EPP6xxxEK1122.A_0006_EPP6002_0002_0018.COM_TxPDO_Map_Inputs_Channel_1.Data_In[7] <-> COM TxPDO-Map Inputs Channel 1/Data In 7
//     PlcTask Inputs/GVL_iXlinker.EtherCAT_Master_EPPxxxx.Beckhoff_EPP6xxx.Beckhoff_EPP6xxxEK1122.A_0006_EPP6002_0002_0018.COM_TxPDO_Map_Inputs_Channel_1.Data_In[8] <-> COM TxPDO-Map Inputs Channel 1/Data In 8
//     PlcTask Inputs/GVL_iXlinker.EtherCAT_Master_EPPxxxx.Beckhoff_EPP6xxx.Beckhoff_EPP6xxxEK1122.A_0006_EPP6002_0002_0018.COM_TxPDO_Map_Inputs_Channel_1.Data_In[9] <-> COM TxPDO-Map Inputs Channel 1/Data In 9
//     PlcTask Inputs/GVL_iXlinker.EtherCAT_Master_EPPxxxx.Beckhoff_EPP6xxx.Beckhoff_EPP6xxxEK1122.A_0006_EPP6002_0002_0018.COM_TxPDO_Map_Inputs_Channel_1.Data_In[10] <-> COM TxPDO-Map Inputs Channel 1/Data In 10
//     PlcTask Inputs/GVL_iXlinker.EtherCAT_Master_EPPxxxx.Beckhoff_EPP6xxx.Beckhoff_EPP6xxxEK1122.A_0006_EPP6002_0002_0018.COM_TxPDO_Map_Inputs_Channel_1.Data_In[11] <-> COM TxPDO-Map Inputs Channel 1/Data In 11
//     PlcTask Inputs/GVL_iXlinker.EtherCAT_Master_EPPxxxx.Beckhoff_EPP6xxx.Beckhoff_EPP6xxxEK1122.A_0006_EPP6002_0002_0018.COM_TxPDO_Map_Inputs_Channel_1.Data_In[12] <-> COM TxPDO-Map Inputs Channel 1/Data In 12
//     PlcTask Inputs/GVL_iXlinker.EtherCAT_Master_EPPxxxx.Beckhoff_EPP6xxx.Beckhoff_EPP6xxxEK1122.A_0006_EPP6002_0002_0018.COM_TxPDO_Map_Inputs_Channel_1.Data_In[13] <-> COM TxPDO-Map Inputs Channel 1/Data In 13
//     PlcTask Inputs/GVL_iXlinker.EtherCAT_Master_EPPxxxx.Beckhoff_EPP6xxx.Beckhoff_EPP6xxxEK1122.A_0006_EPP6002_0002_0018.COM_TxPDO_Map_Inputs_Channel_1.Data_In[14] <-> COM TxPDO-Map Inputs Channel 1/Data In 14
//     PlcTask Inputs/GVL_iXlinker.EtherCAT_Master_EPPxxxx.Beckhoff_EPP6xxx.Beckhoff_EPP6xxxEK1122.A_0006_EPP6002_0002_0018.COM_TxPDO_Map_Inputs_Channel_1.Data_In[15] <-> COM TxPDO-Map Inputs Channel 1/Data In 15
//     PlcTask Inputs/GVL_iXlinker.EtherCAT_Master_EPPxxxx.Beckhoff_EPP6xxx.Beckhoff_EPP6xxxEK1122.A_0006_EPP6002_0002_0018.COM_TxPDO_Map_Inputs_Channel_1.Data_In[16] <-> COM TxPDO-Map Inputs Channel 1/Data In 16
//     PlcTask Inputs/GVL_iXlinker.EtherCAT_Master_EPPxxxx.Beckhoff_EPP6xxx.Beckhoff_EPP6xxxEK1122.A_0006_EPP6002_0002_0018.COM_TxPDO_Map_Inputs_Channel_1.Data_In[17] <-> COM TxPDO-Map Inputs Channel 1/Data In 17
//     PlcTask Inputs/GVL_iXlinker.EtherCAT_Master_EPPxxxx.Beckhoff_EPP6xxx.Beckhoff_EPP6xxxEK1122.A_0006_EPP6002_0002_0018.COM_TxPDO_Map_Inputs_Channel_1.Data_In[18] <-> COM TxPDO-Map Inputs Channel 1/Data In 18
//     PlcTask Inputs/GVL_iXlinker.EtherCAT_Master_EPPxxxx.Beckhoff_EPP6xxx.Beckhoff_EPP6xxxEK1122.A_0006_EPP6002_0002_0018.COM_TxPDO_Map_Inputs_Channel_1.Data_In[19] <-> COM TxPDO-Map Inputs Channel 1/Data In 19
//     PlcTask Inputs/GVL_iXlinker.EtherCAT_Master_EPPxxxx.Beckhoff_EPP6xxx.Beckhoff_EPP6xxxEK1122.A_0006_EPP6002_0002_0018.COM_TxPDO_Map_Inputs_Channel_1.Data_In[20] <-> COM TxPDO-Map Inputs Channel 1/Data In 20
//     PlcTask Inputs/GVL_iXlinker.EtherCAT_Master_EPPxxxx.Beckhoff_EPP6xxx.Beckhoff_EPP6xxxEK1122.A_0006_EPP6002_0002_0018.COM_TxPDO_Map_Inputs_Channel_1.Data_In[21] <-> COM TxPDO-Map Inputs Channel 1/Data In 21
//     PlcTask Inputs/GVL_iXlinker.EtherCAT_Master_EPPxxxx.Beckhoff_EPP6xxx.Beckhoff_EPP6xxxEK1122.A_0006_EPP6002_0002_0018.COM_TxPDO_Map_Inputs_Channel_2.Data_In[0] <-> COM TxPDO-Map Inputs Channel 2/Data In 0
//     PlcTask Inputs/GVL_iXlinker.EtherCAT_Master_EPPxxxx.Beckhoff_EPP6xxx.Beckhoff_EPP6xxxEK1122.A_0006_EPP6002_0002_0018.COM_TxPDO_Map_Inputs_Channel_2.Data_In[1] <-> COM TxPDO-Map Inputs Channel 2/Data In 1
//     PlcTask Inputs/GVL_iXlinker.EtherCAT_Master_EPPxxxx.Beckhoff_EPP6xxx.Beckhoff_EPP6xxxEK1122.A_0006_EPP6002_0002_0018.COM_TxPDO_Map_Inputs_Channel_2.Data_In[2] <-> COM TxPDO-Map Inputs Channel 2/Data In 2
//     PlcTask Inputs/GVL_iXlinker.EtherCAT_Master_EPPxxxx.Beckhoff_EPP6xxx.Beckhoff_EPP6xxxEK1122.A_0006_EPP6002_0002_0018.COM_TxPDO_Map_Inputs_Channel_2.Data_In[3] <-> COM TxPDO-Map Inputs Channel 2/Data In 3
//     PlcTask Inputs/GVL_iXlinker.EtherCAT_Master_EPPxxxx.Beckhoff_EPP6xxx.Beckhoff_EPP6xxxEK1122.A_0006_EPP6002_0002_0018.COM_TxPDO_Map_Inputs_Channel_2.Data_In[4] <-> COM TxPDO-Map Inputs Channel 2/Data In 4
//     PlcTask Inputs/GVL_iXlinker.EtherCAT_Master_EPPxxxx.Beckhoff_EPP6xxx.Beckhoff_EPP6xxxEK1122.A_0006_EPP6002_0002_0018.COM_TxPDO_Map_Inputs_Channel_2.Data_In[5] <-> COM TxPDO-Map Inputs Channel 2/Data In 5
//     PlcTask Inputs/GVL_iXlinker.EtherCAT_Master_EPPxxxx.Beckhoff_EPP6xxx.Beckhoff_EPP6xxxEK1122.A_0006_EPP6002_0002_0018.COM_TxPDO_Map_Inputs_Channel_2.Data_In[6] <-> COM TxPDO-Map Inputs Channel 2/Data In 6
//     PlcTask Inputs/GVL_iXlinker.EtherCAT_Master_EPPxxxx.Beckhoff_EPP6xxx.Beckhoff_EPP6xxxEK1122.A_0006_EPP6002_0002_0018.COM_TxPDO_Map_Inputs_Channel_2.Data_In[7] <-> COM TxPDO-Map Inputs Channel 2/Data In 7
//     PlcTask Inputs/GVL_iXlinker.EtherCAT_Master_EPPxxxx.Beckhoff_EPP6xxx.Beckhoff_EPP6xxxEK1122.A_0006_EPP6002_0002_0018.COM_TxPDO_Map_Inputs_Channel_2.Data_In[8] <-> COM TxPDO-Map Inputs Channel 2/Data In 8
//     PlcTask Inputs/GVL_iXlinker.EtherCAT_Master_EPPxxxx.Beckhoff_EPP6xxx.Beckhoff_EPP6xxxEK1122.A_0006_EPP6002_0002_0018.COM_TxPDO_Map_Inputs_Channel_2.Data_In[9] <-> COM TxPDO-Map Inputs Channel 2/Data In 9
//     PlcTask Inputs/GVL_iXlinker.EtherCAT_Master_EPPxxxx.Beckhoff_EPP6xxx.Beckhoff_EPP6xxxEK1122.A_0006_EPP6002_0002_0018.COM_TxPDO_Map_Inputs_Channel_2.Data_In[10] <-> COM TxPDO-Map Inputs Channel 2/Data In 10
//     PlcTask Inputs/GVL_iXlinker.EtherCAT_Master_EPPxxxx.Beckhoff_EPP6xxx.Beckhoff_EPP6xxxEK1122.A_0006_EPP6002_0002_0018.COM_TxPDO_Map_Inputs_Channel_2.Data_In[11] <-> COM TxPDO-Map Inputs Channel 2/Data In 11
//     PlcTask Inputs/GVL_iXlinker.EtherCAT_Master_EPPxxxx.Beckhoff_EPP6xxx.Beckhoff_EPP6xxxEK1122.A_0006_EPP6002_0002_0018.COM_TxPDO_Map_Inputs_Channel_2.Data_In[12] <-> COM TxPDO-Map Inputs Channel 2/Data In 12
//     PlcTask Inputs/GVL_iXlinker.EtherCAT_Master_EPPxxxx.Beckhoff_EPP6xxx.Beckhoff_EPP6xxxEK1122.A_0006_EPP6002_0002_0018.COM_TxPDO_Map_Inputs_Channel_2.Data_In[13] <-> COM TxPDO-Map Inputs Channel 2/Data In 13
//     PlcTask Inputs/GVL_iXlinker.EtherCAT_Master_EPPxxxx.Beckhoff_EPP6xxx.Beckhoff_EPP6xxxEK1122.A_0006_EPP6002_0002_0018.COM_TxPDO_Map_Inputs_Channel_2.Data_In[14] <-> COM TxPDO-Map Inputs Channel 2/Data In 14
//     PlcTask Inputs/GVL_iXlinker.EtherCAT_Master_EPPxxxx.Beckhoff_EPP6xxx.Beckhoff_EPP6xxxEK1122.A_0006_EPP6002_0002_0018.COM_TxPDO_Map_Inputs_Channel_2.Data_In[15] <-> COM TxPDO-Map Inputs Channel 2/Data In 15
//     PlcTask Inputs/GVL_iXlinker.EtherCAT_Master_EPPxxxx.Beckhoff_EPP6xxx.Beckhoff_EPP6xxxEK1122.A_0006_EPP6002_0002_0018.COM_TxPDO_Map_Inputs_Channel_2.Data_In[16] <-> COM TxPDO-Map Inputs Channel 2/Data In 16
//     PlcTask Inputs/GVL_iXlinker.EtherCAT_Master_EPPxxxx.Beckhoff_EPP6xxx.Beckhoff_EPP6xxxEK1122.A_0006_EPP6002_0002_0018.COM_TxPDO_Map_Inputs_Channel_2.Data_In[17] <-> COM TxPDO-Map Inputs Channel 2/Data In 17
//     PlcTask Inputs/GVL_iXlinker.EtherCAT_Master_EPPxxxx.Beckhoff_EPP6xxx.Beckhoff_EPP6xxxEK1122.A_0006_EPP6002_0002_0018.COM_TxPDO_Map_Inputs_Channel_2.Data_In[18] <-> COM TxPDO-Map Inputs Channel 2/Data In 18
//     PlcTask Inputs/GVL_iXlinker.EtherCAT_Master_EPPxxxx.Beckhoff_EPP6xxx.Beckhoff_EPP6xxxEK1122.A_0006_EPP6002_0002_0018.COM_TxPDO_Map_Inputs_Channel_2.Data_In[19] <-> COM TxPDO-Map Inputs Channel 2/Data In 19
//     PlcTask Inputs/GVL_iXlinker.EtherCAT_Master_EPPxxxx.Beckhoff_EPP6xxx.Beckhoff_EPP6xxxEK1122.A_0006_EPP6002_0002_0018.COM_TxPDO_Map_Inputs_Channel_2.Data_In[20] <-> COM TxPDO-Map Inputs Channel 2/Data In 20
//     PlcTask Inputs/GVL_iXlinker.EtherCAT_Master_EPPxxxx.Beckhoff_EPP6xxx.Beckhoff_EPP6xxxEK1122.A_0006_EPP6002_0002_0018.COM_TxPDO_Map_Inputs_Channel_2.Data_In[21] <-> COM TxPDO-Map Inputs Channel 2/Data In 21
//     PlcTask Outputs/GVL_iXlinker.EtherCAT_Master_EPPxxxx.Beckhoff_EPP6xxx.Beckhoff_EPP6xxxEK1122.A_0006_EPP6002_0002_0018.COM_RxPDO_Map_Outputs_Channel_1.Ctrl <-> COM RxPDO-Map Outputs Channel 1/Ctrl
//     PlcTask Outputs/GVL_iXlinker.EtherCAT_Master_EPPxxxx.Beckhoff_EPP6xxx.Beckhoff_EPP6xxxEK1122.A_0006_EPP6002_0002_0018.COM_RxPDO_Map_Outputs_Channel_2.Ctrl <-> COM RxPDO-Map Outputs Channel 2/Ctrl
//     PlcTask Outputs/GVL_iXlinker.EtherCAT_Master_EPPxxxx.Beckhoff_EPP6xxx.Beckhoff_EPP6xxxEK1122.A_0006_EPP6002_0002_0018.COM_RxPDO_Map_Outputs_Channel_1.Data_Out[0] <-> COM RxPDO-Map Outputs Channel 1/Data Out 0
//     PlcTask Outputs/GVL_iXlinker.EtherCAT_Master_EPPxxxx.Beckhoff_EPP6xxx.Beckhoff_EPP6xxxEK1122.A_0006_EPP6002_0002_0018.COM_RxPDO_Map_Outputs_Channel_1.Data_Out[1] <-> COM RxPDO-Map Outputs Channel 1/Data Out 1
//     PlcTask Outputs/GVL_iXlinker.EtherCAT_Master_EPPxxxx.Beckhoff_EPP6xxx.Beckhoff_EPP6xxxEK1122.A_0006_EPP6002_0002_0018.COM_RxPDO_Map_Outputs_Channel_1.Data_Out[2] <-> COM RxPDO-Map Outputs Channel 1/Data Out 2
//     PlcTask Outputs/GVL_iXlinker.EtherCAT_Master_EPPxxxx.Beckhoff_EPP6xxx.Beckhoff_EPP6xxxEK1122.A_0006_EPP6002_0002_0018.COM_RxPDO_Map_Outputs_Channel_1.Data_Out[3] <-> COM RxPDO-Map Outputs Channel 1/Data Out 3
//     PlcTask Outputs/GVL_iXlinker.EtherCAT_Master_EPPxxxx.Beckhoff_EPP6xxx.Beckhoff_EPP6xxxEK1122.A_0006_EPP6002_0002_0018.COM_RxPDO_Map_Outputs_Channel_1.Data_Out[4] <-> COM RxPDO-Map Outputs Channel 1/Data Out 4
//     PlcTask Outputs/GVL_iXlinker.EtherCAT_Master_EPPxxxx.Beckhoff_EPP6xxx.Beckhoff_EPP6xxxEK1122.A_0006_EPP6002_0002_0018.COM_RxPDO_Map_Outputs_Channel_1.Data_Out[5] <-> COM RxPDO-Map Outputs Channel 1/Data Out 5
//     PlcTask Outputs/GVL_iXlinker.EtherCAT_Master_EPPxxxx.Beckhoff_EPP6xxx.Beckhoff_EPP6xxxEK1122.A_0006_EPP6002_0002_0018.COM_RxPDO_Map_Outputs_Channel_1.Data_Out[6] <-> COM RxPDO-Map Outputs Channel 1/Data Out 6
//     PlcTask Outputs/GVL_iXlinker.EtherCAT_Master_EPPxxxx.Beckhoff_EPP6xxx.Beckhoff_EPP6xxxEK1122.A_0006_EPP6002_0002_0018.COM_RxPDO_Map_Outputs_Channel_1.Data_Out[7] <-> COM RxPDO-Map Outputs Channel 1/Data Out 7
//     PlcTask Outputs/GVL_iXlinker.EtherCAT_Master_EPPxxxx.Beckhoff_EPP6xxx.Beckhoff_EPP6xxxEK1122.A_0006_EPP6002_0002_0018.COM_RxPDO_Map_Outputs_Channel_1.Data_Out[8] <-> COM RxPDO-Map Outputs Channel 1/Data Out 8
//     PlcTask Outputs/GVL_iXlinker.EtherCAT_Master_EPPxxxx.Beckhoff_EPP6xxx.Beckhoff_EPP6xxxEK1122.A_0006_EPP6002_0002_0018.COM_RxPDO_Map_Outputs_Channel_1.Data_Out[9] <-> COM RxPDO-Map Outputs Channel 1/Data Out 9
//     PlcTask Outputs/GVL_iXlinker.EtherCAT_Master_EPPxxxx.Beckhoff_EPP6xxx.Beckhoff_EPP6xxxEK1122.A_0006_EPP6002_0002_0018.COM_RxPDO_Map_Outputs_Channel_1.Data_Out[10] <-> COM RxPDO-Map Outputs Channel 1/Data Out 10
//     PlcTask Outputs/GVL_iXlinker.EtherCAT_Master_EPPxxxx.Beckhoff_EPP6xxx.Beckhoff_EPP6xxxEK1122.A_0006_EPP6002_0002_0018.COM_RxPDO_Map_Outputs_Channel_1.Data_Out[11] <-> COM RxPDO-Map Outputs Channel 1/Data Out 11
//     PlcTask Outputs/GVL_iXlinker.EtherCAT_Master_EPPxxxx.Beckhoff_EPP6xxx.Beckhoff_EPP6xxxEK1122.A_0006_EPP6002_0002_0018.COM_RxPDO_Map_Outputs_Channel_1.Data_Out[12] <-> COM RxPDO-Map Outputs Channel 1/Data Out 12
//     PlcTask Outputs/GVL_iXlinker.EtherCAT_Master_EPPxxxx.Beckhoff_EPP6xxx.Beckhoff_EPP6xxxEK1122.A_0006_EPP6002_0002_0018.COM_RxPDO_Map_Outputs_Channel_1.Data_Out[13] <-> COM RxPDO-Map Outputs Channel 1/Data Out 13
//     PlcTask Outputs/GVL_iXlinker.EtherCAT_Master_EPPxxxx.Beckhoff_EPP6xxx.Beckhoff_EPP6xxxEK1122.A_0006_EPP6002_0002_0018.COM_RxPDO_Map_Outputs_Channel_1.Data_Out[14] <-> COM RxPDO-Map Outputs Channel 1/Data Out 14
//     PlcTask Outputs/GVL_iXlinker.EtherCAT_Master_EPPxxxx.Beckhoff_EPP6xxx.Beckhoff_EPP6xxxEK1122.A_0006_EPP6002_0002_0018.COM_RxPDO_Map_Outputs_Channel_1.Data_Out[15] <-> COM RxPDO-Map Outputs Channel 1/Data Out 15
//     PlcTask Outputs/GVL_iXlinker.EtherCAT_Master_EPPxxxx.Beckhoff_EPP6xxx.Beckhoff_EPP6xxxEK1122.A_0006_EPP6002_0002_0018.COM_RxPDO_Map_Outputs_Channel_1.Data_Out[16] <-> COM RxPDO-Map Outputs Channel 1/Data Out 16
//     PlcTask Outputs/GVL_iXlinker.EtherCAT_Master_EPPxxxx.Beckhoff_EPP6xxx.Beckhoff_EPP6xxxEK1122.A_0006_EPP6002_0002_0018.COM_RxPDO_Map_Outputs_Channel_1.Data_Out[17] <-> COM RxPDO-Map Outputs Channel 1/Data Out 17
//     PlcTask Outputs/GVL_iXlinker.EtherCAT_Master_EPPxxxx.Beckhoff_EPP6xxx.Beckhoff_EPP6xxxEK1122.A_0006_EPP6002_0002_0018.COM_RxPDO_Map_Outputs_Channel_1.Data_Out[18] <-> COM RxPDO-Map Outputs Channel 1/Data Out 18
//     PlcTask Outputs/GVL_iXlinker.EtherCAT_Master_EPPxxxx.Beckhoff_EPP6xxx.Beckhoff_EPP6xxxEK1122.A_0006_EPP6002_0002_0018.COM_RxPDO_Map_Outputs_Channel_1.Data_Out[19] <-> COM RxPDO-Map Outputs Channel 1/Data Out 19
//     PlcTask Outputs/GVL_iXlinker.EtherCAT_Master_EPPxxxx.Beckhoff_EPP6xxx.Beckhoff_EPP6xxxEK1122.A_0006_EPP6002_0002_0018.COM_RxPDO_Map_Outputs_Channel_1.Data_Out[20] <-> COM RxPDO-Map Outputs Channel 1/Data Out 20
//     PlcTask Outputs/GVL_iXlinker.EtherCAT_Master_EPPxxxx.Beckhoff_EPP6xxx.Beckhoff_EPP6xxxEK1122.A_0006_EPP6002_0002_0018.COM_RxPDO_Map_Outputs_Channel_1.Data_Out[21] <-> COM RxPDO-Map Outputs Channel 1/Data Out 21
//     PlcTask Outputs/GVL_iXlinker.EtherCAT_Master_EPPxxxx.Beckhoff_EPP6xxx.Beckhoff_EPP6xxxEK1122.A_0006_EPP6002_0002_0018.COM_RxPDO_Map_Outputs_Channel_2.Data_Out[0] <-> COM RxPDO-Map Outputs Channel 2/Data Out 0
//     PlcTask Outputs/GVL_iXlinker.EtherCAT_Master_EPPxxxx.Beckhoff_EPP6xxx.Beckhoff_EPP6xxxEK1122.A_0006_EPP6002_0002_0018.COM_RxPDO_Map_Outputs_Channel_2.Data_Out[1] <-> COM RxPDO-Map Outputs Channel 2/Data Out 1
//     PlcTask Outputs/GVL_iXlinker.EtherCAT_Master_EPPxxxx.Beckhoff_EPP6xxx.Beckhoff_EPP6xxxEK1122.A_0006_EPP6002_0002_0018.COM_RxPDO_Map_Outputs_Channel_2.Data_Out[2] <-> COM RxPDO-Map Outputs Channel 2/Data Out 2
//     PlcTask Outputs/GVL_iXlinker.EtherCAT_Master_EPPxxxx.Beckhoff_EPP6xxx.Beckhoff_EPP6xxxEK1122.A_0006_EPP6002_0002_0018.COM_RxPDO_Map_Outputs_Channel_2.Data_Out[3] <-> COM RxPDO-Map Outputs Channel 2/Data Out 3
//     PlcTask Outputs/GVL_iXlinker.EtherCAT_Master_EPPxxxx.Beckhoff_EPP6xxx.Beckhoff_EPP6xxxEK1122.A_0006_EPP6002_0002_0018.COM_RxPDO_Map_Outputs_Channel_2.Data_Out[4] <-> COM RxPDO-Map Outputs Channel 2/Data Out 4
//     PlcTask Outputs/GVL_iXlinker.EtherCAT_Master_EPPxxxx.Beckhoff_EPP6xxx.Beckhoff_EPP6xxxEK1122.A_0006_EPP6002_0002_0018.COM_RxPDO_Map_Outputs_Channel_2.Data_Out[5] <-> COM RxPDO-Map Outputs Channel 2/Data Out 5
//     PlcTask Outputs/GVL_iXlinker.EtherCAT_Master_EPPxxxx.Beckhoff_EPP6xxx.Beckhoff_EPP6xxxEK1122.A_0006_EPP6002_0002_0018.COM_RxPDO_Map_Outputs_Channel_2.Data_Out[6] <-> COM RxPDO-Map Outputs Channel 2/Data Out 6
//     PlcTask Outputs/GVL_iXlinker.EtherCAT_Master_EPPxxxx.Beckhoff_EPP6xxx.Beckhoff_EPP6xxxEK1122.A_0006_EPP6002_0002_0018.COM_RxPDO_Map_Outputs_Channel_2.Data_Out[7] <-> COM RxPDO-Map Outputs Channel 2/Data Out 7
//     PlcTask Outputs/GVL_iXlinker.EtherCAT_Master_EPPxxxx.Beckhoff_EPP6xxx.Beckhoff_EPP6xxxEK1122.A_0006_EPP6002_0002_0018.COM_RxPDO_Map_Outputs_Channel_2.Data_Out[8] <-> COM RxPDO-Map Outputs Channel 2/Data Out 8
//     PlcTask Outputs/GVL_iXlinker.EtherCAT_Master_EPPxxxx.Beckhoff_EPP6xxx.Beckhoff_EPP6xxxEK1122.A_0006_EPP6002_0002_0018.COM_RxPDO_Map_Outputs_Channel_2.Data_Out[9] <-> COM RxPDO-Map Outputs Channel 2/Data Out 9
//     PlcTask Outputs/GVL_iXlinker.EtherCAT_Master_EPPxxxx.Beckhoff_EPP6xxx.Beckhoff_EPP6xxxEK1122.A_0006_EPP6002_0002_0018.COM_RxPDO_Map_Outputs_Channel_2.Data_Out[10] <-> COM RxPDO-Map Outputs Channel 2/Data Out 10
//     PlcTask Outputs/GVL_iXlinker.EtherCAT_Master_EPPxxxx.Beckhoff_EPP6xxx.Beckhoff_EPP6xxxEK1122.A_0006_EPP6002_0002_0018.COM_RxPDO_Map_Outputs_Channel_2.Data_Out[11] <-> COM RxPDO-Map Outputs Channel 2/Data Out 11
//     PlcTask Outputs/GVL_iXlinker.EtherCAT_Master_EPPxxxx.Beckhoff_EPP6xxx.Beckhoff_EPP6xxxEK1122.A_0006_EPP6002_0002_0018.COM_RxPDO_Map_Outputs_Channel_2.Data_Out[12] <-> COM RxPDO-Map Outputs Channel 2/Data Out 12
//     PlcTask Outputs/GVL_iXlinker.EtherCAT_Master_EPPxxxx.Beckhoff_EPP6xxx.Beckhoff_EPP6xxxEK1122.A_0006_EPP6002_0002_0018.COM_RxPDO_Map_Outputs_Channel_2.Data_Out[13] <-> COM RxPDO-Map Outputs Channel 2/Data Out 13
//     PlcTask Outputs/GVL_iXlinker.EtherCAT_Master_EPPxxxx.Beckhoff_EPP6xxx.Beckhoff_EPP6xxxEK1122.A_0006_EPP6002_0002_0018.COM_RxPDO_Map_Outputs_Channel_2.Data_Out[14] <-> COM RxPDO-Map Outputs Channel 2/Data Out 14
//     PlcTask Outputs/GVL_iXlinker.EtherCAT_Master_EPPxxxx.Beckhoff_EPP6xxx.Beckhoff_EPP6xxxEK1122.A_0006_EPP6002_0002_0018.COM_RxPDO_Map_Outputs_Channel_2.Data_Out[15] <-> COM RxPDO-Map Outputs Channel 2/Data Out 15
//     PlcTask Outputs/GVL_iXlinker.EtherCAT_Master_EPPxxxx.Beckhoff_EPP6xxx.Beckhoff_EPP6xxxEK1122.A_0006_EPP6002_0002_0018.COM_RxPDO_Map_Outputs_Channel_2.Data_Out[16] <-> COM RxPDO-Map Outputs Channel 2/Data Out 16
//     PlcTask Outputs/GVL_iXlinker.EtherCAT_Master_EPPxxxx.Beckhoff_EPP6xxx.Beckhoff_EPP6xxxEK1122.A_0006_EPP6002_0002_0018.COM_RxPDO_Map_Outputs_Channel_2.Data_Out[17] <-> COM RxPDO-Map Outputs Channel 2/Data Out 17
//     PlcTask Outputs/GVL_iXlinker.EtherCAT_Master_EPPxxxx.Beckhoff_EPP6xxx.Beckhoff_EPP6xxxEK1122.A_0006_EPP6002_0002_0018.COM_RxPDO_Map_Outputs_Channel_2.Data_Out[18] <-> COM RxPDO-Map Outputs Channel 2/Data Out 18
//     PlcTask Outputs/GVL_iXlinker.EtherCAT_Master_EPPxxxx.Beckhoff_EPP6xxx.Beckhoff_EPP6xxxEK1122.A_0006_EPP6002_0002_0018.COM_RxPDO_Map_Outputs_Channel_2.Data_Out[19] <-> COM RxPDO-Map Outputs Channel 2/Data Out 19
//     PlcTask Outputs/GVL_iXlinker.EtherCAT_Master_EPPxxxx.Beckhoff_EPP6xxx.Beckhoff_EPP6xxxEK1122.A_0006_EPP6002_0002_0018.COM_RxPDO_Map_Outputs_Channel_2.Data_Out[20] <-> COM RxPDO-Map Outputs Channel 2/Data Out 20
//     PlcTask Outputs/GVL_iXlinker.EtherCAT_Master_EPPxxxx.Beckhoff_EPP6xxx.Beckhoff_EPP6xxxEK1122.A_0006_EPP6002_0002_0018.COM_RxPDO_Map_Outputs_Channel_2.Data_Out[21] <-> COM RxPDO-Map Outputs Channel 2/Data Out 21
//     PlcTask Inputs/GVL_iXlinker.EtherCAT_Master_EPPxxxx.Beckhoff_EPP6xxx.Beckhoff_EPP6xxxEK1122.A_0006_EPP6002_0002_0018.WcState.WcState <-> WcState/WcState
//     PlcTask Inputs/GVL_iXlinker.EtherCAT_Master_EPPxxxx.Beckhoff_EPP6xxx.Beckhoff_EPP6xxxEK1122.A_0006_EPP6002_0002_0018.WcState.InputToggle <-> WcState/InputToggle
//     PlcTask Inputs/GVL_iXlinker.EtherCAT_Master_EPPxxxx.Beckhoff_EPP6xxx.Beckhoff_EPP6xxxEK1122.A_0006_EPP6002_0002_0018.InfoData.AdsAddr <-> InfoData/AdsAddr
//     PlcTask Inputs/GVL_iXlinker.EtherCAT_Master_EPPxxxx.Beckhoff_EPP6xxx.Beckhoff_EPP6xxxEK1122.A_0006_EPP6002_0002_0018.InfoData.State <-> InfoData/State
//   PLC/PLC Instance <-> EtherCAT Master EPPxxxx/Beckhoff EPP6xxx/Beckhoff EPP6xxxEK1122/A_0007(EPP6002-0002-0019)
//     PlcTask Inputs/GVL_iXlinker.EtherCAT_Master_EPPxxxx.Beckhoff_EPP6xxx.Beckhoff_EPP6xxxEK1122.A_0007_EPP6002_0002_0019.COM_TxPDO_Map_Inputs_Channel_1.Status <-> COM TxPDO-Map Inputs Channel 1/Status
//     PlcTask Inputs/GVL_iXlinker.EtherCAT_Master_EPPxxxx.Beckhoff_EPP6xxx.Beckhoff_EPP6xxxEK1122.A_0007_EPP6002_0002_0019.COM_TxPDO_Map_Inputs_Channel_2.Status <-> COM TxPDO-Map Inputs Channel 2/Status
//     PlcTask Inputs/GVL_iXlinker.EtherCAT_Master_EPPxxxx.Beckhoff_EPP6xxx.Beckhoff_EPP6xxxEK1122.A_0007_EPP6002_0002_0019.COM_TxPDO_Map_Inputs_Channel_1.Data_In[0] <-> COM TxPDO-Map Inputs Channel 1/Data In 0
//     PlcTask Inputs/GVL_iXlinker.EtherCAT_Master_EPPxxxx.Beckhoff_EPP6xxx.Beckhoff_EPP6xxxEK1122.A_0007_EPP6002_0002_0019.COM_TxPDO_Map_Inputs_Channel_1.Data_In[1] <-> COM TxPDO-Map Inputs Channel 1/Data In 1
//     PlcTask Inputs/GVL_iXlinker.EtherCAT_Master_EPPxxxx.Beckhoff_EPP6xxx.Beckhoff_EPP6xxxEK1122.A_0007_EPP6002_0002_0019.COM_TxPDO_Map_Inputs_Channel_1.Data_In[2] <-> COM TxPDO-Map Inputs Channel 1/Data In 2
//     PlcTask Inputs/GVL_iXlinker.EtherCAT_Master_EPPxxxx.Beckhoff_EPP6xxx.Beckhoff_EPP6xxxEK1122.A_0007_EPP6002_0002_0019.COM_TxPDO_Map_Inputs_Channel_1.Data_In[3] <-> COM TxPDO-Map Inputs Channel 1/Data In 3
//     PlcTask Inputs/GVL_iXlinker.EtherCAT_Master_EPPxxxx.Beckhoff_EPP6xxx.Beckhoff_EPP6xxxEK1122.A_0007_EPP6002_0002_0019.COM_TxPDO_Map_Inputs_Channel_1.Data_In[4] <-> COM TxPDO-Map Inputs Channel 1/Data In 4
//     PlcTask Inputs/GVL_iXlinker.EtherCAT_Master_EPPxxxx.Beckhoff_EPP6xxx.Beckhoff_EPP6xxxEK1122.A_0007_EPP6002_0002_0019.COM_TxPDO_Map_Inputs_Channel_1.Data_In[5] <-> COM TxPDO-Map Inputs Channel 1/Data In 5
//     PlcTask Inputs/GVL_iXlinker.EtherCAT_Master_EPPxxxx.Beckhoff_EPP6xxx.Beckhoff_EPP6xxxEK1122.A_0007_EPP6002_0002_0019.COM_TxPDO_Map_Inputs_Channel_1.Data_In[6] <-> COM TxPDO-Map Inputs Channel 1/Data In 6
//     PlcTask Inputs/GVL_iXlinker.EtherCAT_Master_EPPxxxx.Beckhoff_EPP6xxx.Beckhoff_EPP6xxxEK1122.A_0007_EPP6002_0002_0019.COM_TxPDO_Map_Inputs_Channel_1.Data_In[7] <-> COM TxPDO-Map Inputs Channel 1/Data In 7
//     PlcTask Inputs/GVL_iXlinker.EtherCAT_Master_EPPxxxx.Beckhoff_EPP6xxx.Beckhoff_EPP6xxxEK1122.A_0007_EPP6002_0002_0019.COM_TxPDO_Map_Inputs_Channel_1.Data_In[8] <-> COM TxPDO-Map Inputs Channel 1/Data In 8
//     PlcTask Inputs/GVL_iXlinker.EtherCAT_Master_EPPxxxx.Beckhoff_EPP6xxx.Beckhoff_EPP6xxxEK1122.A_0007_EPP6002_0002_0019.COM_TxPDO_Map_Inputs_Channel_1.Data_In[9] <-> COM TxPDO-Map Inputs Channel 1/Data In 9
//     PlcTask Inputs/GVL_iXlinker.EtherCAT_Master_EPPxxxx.Beckhoff_EPP6xxx.Beckhoff_EPP6xxxEK1122.A_0007_EPP6002_0002_0019.COM_TxPDO_Map_Inputs_Channel_1.Data_In[10] <-> COM TxPDO-Map Inputs Channel 1/Data In 10
//     PlcTask Inputs/GVL_iXlinker.EtherCAT_Master_EPPxxxx.Beckhoff_EPP6xxx.Beckhoff_EPP6xxxEK1122.A_0007_EPP6002_0002_0019.COM_TxPDO_Map_Inputs_Channel_1.Data_In[11] <-> COM TxPDO-Map Inputs Channel 1/Data In 11
//     PlcTask Inputs/GVL_iXlinker.EtherCAT_Master_EPPxxxx.Beckhoff_EPP6xxx.Beckhoff_EPP6xxxEK1122.A_0007_EPP6002_0002_0019.COM_TxPDO_Map_Inputs_Channel_1.Data_In[12] <-> COM TxPDO-Map Inputs Channel 1/Data In 12
//     PlcTask Inputs/GVL_iXlinker.EtherCAT_Master_EPPxxxx.Beckhoff_EPP6xxx.Beckhoff_EPP6xxxEK1122.A_0007_EPP6002_0002_0019.COM_TxPDO_Map_Inputs_Channel_1.Data_In[13] <-> COM TxPDO-Map Inputs Channel 1/Data In 13
//     PlcTask Inputs/GVL_iXlinker.EtherCAT_Master_EPPxxxx.Beckhoff_EPP6xxx.Beckhoff_EPP6xxxEK1122.A_0007_EPP6002_0002_0019.COM_TxPDO_Map_Inputs_Channel_1.Data_In[14] <-> COM TxPDO-Map Inputs Channel 1/Data In 14
//     PlcTask Inputs/GVL_iXlinker.EtherCAT_Master_EPPxxxx.Beckhoff_EPP6xxx.Beckhoff_EPP6xxxEK1122.A_0007_EPP6002_0002_0019.COM_TxPDO_Map_Inputs_Channel_1.Data_In[15] <-> COM TxPDO-Map Inputs Channel 1/Data In 15
//     PlcTask Inputs/GVL_iXlinker.EtherCAT_Master_EPPxxxx.Beckhoff_EPP6xxx.Beckhoff_EPP6xxxEK1122.A_0007_EPP6002_0002_0019.COM_TxPDO_Map_Inputs_Channel_1.Data_In[16] <-> COM TxPDO-Map Inputs Channel 1/Data In 16
//     PlcTask Inputs/GVL_iXlinker.EtherCAT_Master_EPPxxxx.Beckhoff_EPP6xxx.Beckhoff_EPP6xxxEK1122.A_0007_EPP6002_0002_0019.COM_TxPDO_Map_Inputs_Channel_1.Data_In[17] <-> COM TxPDO-Map Inputs Channel 1/Data In 17
//     PlcTask Inputs/GVL_iXlinker.EtherCAT_Master_EPPxxxx.Beckhoff_EPP6xxx.Beckhoff_EPP6xxxEK1122.A_0007_EPP6002_0002_0019.COM_TxPDO_Map_Inputs_Channel_1.Data_In[18] <-> COM TxPDO-Map Inputs Channel 1/Data In 18
//     PlcTask Inputs/GVL_iXlinker.EtherCAT_Master_EPPxxxx.Beckhoff_EPP6xxx.Beckhoff_EPP6xxxEK1122.A_0007_EPP6002_0002_0019.COM_TxPDO_Map_Inputs_Channel_1.Data_In[19] <-> COM TxPDO-Map Inputs Channel 1/Data In 19
//     PlcTask Inputs/GVL_iXlinker.EtherCAT_Master_EPPxxxx.Beckhoff_EPP6xxx.Beckhoff_EPP6xxxEK1122.A_0007_EPP6002_0002_0019.COM_TxPDO_Map_Inputs_Channel_1.Data_In[20] <-> COM TxPDO-Map Inputs Channel 1/Data In 20
//     PlcTask Inputs/GVL_iXlinker.EtherCAT_Master_EPPxxxx.Beckhoff_EPP6xxx.Beckhoff_EPP6xxxEK1122.A_0007_EPP6002_0002_0019.COM_TxPDO_Map_Inputs_Channel_1.Data_In[21] <-> COM TxPDO-Map Inputs Channel 1/Data In 21
//     PlcTask Inputs/GVL_iXlinker.EtherCAT_Master_EPPxxxx.Beckhoff_EPP6xxx.Beckhoff_EPP6xxxEK1122.A_0007_EPP6002_0002_0019.COM_TxPDO_Map_Inputs_Channel_2.Data_In[0] <-> COM TxPDO-Map Inputs Channel 2/Data In 0
//     PlcTask Inputs/GVL_iXlinker.EtherCAT_Master_EPPxxxx.Beckhoff_EPP6xxx.Beckhoff_EPP6xxxEK1122.A_0007_EPP6002_0002_0019.COM_TxPDO_Map_Inputs_Channel_2.Data_In[1] <-> COM TxPDO-Map Inputs Channel 2/Data In 1
//     PlcTask Inputs/GVL_iXlinker.EtherCAT_Master_EPPxxxx.Beckhoff_EPP6xxx.Beckhoff_EPP6xxxEK1122.A_0007_EPP6002_0002_0019.COM_TxPDO_Map_Inputs_Channel_2.Data_In[2] <-> COM TxPDO-Map Inputs Channel 2/Data In 2
//     PlcTask Inputs/GVL_iXlinker.EtherCAT_Master_EPPxxxx.Beckhoff_EPP6xxx.Beckhoff_EPP6xxxEK1122.A_0007_EPP6002_0002_0019.COM_TxPDO_Map_Inputs_Channel_2.Data_In[3] <-> COM TxPDO-Map Inputs Channel 2/Data In 3
//     PlcTask Inputs/GVL_iXlinker.EtherCAT_Master_EPPxxxx.Beckhoff_EPP6xxx.Beckhoff_EPP6xxxEK1122.A_0007_EPP6002_0002_0019.COM_TxPDO_Map_Inputs_Channel_2.Data_In[4] <-> COM TxPDO-Map Inputs Channel 2/Data In 4
//     PlcTask Inputs/GVL_iXlinker.EtherCAT_Master_EPPxxxx.Beckhoff_EPP6xxx.Beckhoff_EPP6xxxEK1122.A_0007_EPP6002_0002_0019.COM_TxPDO_Map_Inputs_Channel_2.Data_In[5] <-> COM TxPDO-Map Inputs Channel 2/Data In 5
//     PlcTask Inputs/GVL_iXlinker.EtherCAT_Master_EPPxxxx.Beckhoff_EPP6xxx.Beckhoff_EPP6xxxEK1122.A_0007_EPP6002_0002_0019.COM_TxPDO_Map_Inputs_Channel_2.Data_In[6] <-> COM TxPDO-Map Inputs Channel 2/Data In 6
//     PlcTask Inputs/GVL_iXlinker.EtherCAT_Master_EPPxxxx.Beckhoff_EPP6xxx.Beckhoff_EPP6xxxEK1122.A_0007_EPP6002_0002_0019.COM_TxPDO_Map_Inputs_Channel_2.Data_In[7] <-> COM TxPDO-Map Inputs Channel 2/Data In 7
//     PlcTask Inputs/GVL_iXlinker.EtherCAT_Master_EPPxxxx.Beckhoff_EPP6xxx.Beckhoff_EPP6xxxEK1122.A_0007_EPP6002_0002_0019.COM_TxPDO_Map_Inputs_Channel_2.Data_In[8] <-> COM TxPDO-Map Inputs Channel 2/Data In 8
//     PlcTask Inputs/GVL_iXlinker.EtherCAT_Master_EPPxxxx.Beckhoff_EPP6xxx.Beckhoff_EPP6xxxEK1122.A_0007_EPP6002_0002_0019.COM_TxPDO_Map_Inputs_Channel_2.Data_In[9] <-> COM TxPDO-Map Inputs Channel 2/Data In 9
//     PlcTask Inputs/GVL_iXlinker.EtherCAT_Master_EPPxxxx.Beckhoff_EPP6xxx.Beckhoff_EPP6xxxEK1122.A_0007_EPP6002_0002_0019.COM_TxPDO_Map_Inputs_Channel_2.Data_In[10] <-> COM TxPDO-Map Inputs Channel 2/Data In 10
//     PlcTask Inputs/GVL_iXlinker.EtherCAT_Master_EPPxxxx.Beckhoff_EPP6xxx.Beckhoff_EPP6xxxEK1122.A_0007_EPP6002_0002_0019.COM_TxPDO_Map_Inputs_Channel_2.Data_In[11] <-> COM TxPDO-Map Inputs Channel 2/Data In 11
//     PlcTask Inputs/GVL_iXlinker.EtherCAT_Master_EPPxxxx.Beckhoff_EPP6xxx.Beckhoff_EPP6xxxEK1122.A_0007_EPP6002_0002_0019.COM_TxPDO_Map_Inputs_Channel_2.Data_In[12] <-> COM TxPDO-Map Inputs Channel 2/Data In 12
//     PlcTask Inputs/GVL_iXlinker.EtherCAT_Master_EPPxxxx.Beckhoff_EPP6xxx.Beckhoff_EPP6xxxEK1122.A_0007_EPP6002_0002_0019.COM_TxPDO_Map_Inputs_Channel_2.Data_In[13] <-> COM TxPDO-Map Inputs Channel 2/Data In 13
//     PlcTask Inputs/GVL_iXlinker.EtherCAT_Master_EPPxxxx.Beckhoff_EPP6xxx.Beckhoff_EPP6xxxEK1122.A_0007_EPP6002_0002_0019.COM_TxPDO_Map_Inputs_Channel_2.Data_In[14] <-> COM TxPDO-Map Inputs Channel 2/Data In 14
//     PlcTask Inputs/GVL_iXlinker.EtherCAT_Master_EPPxxxx.Beckhoff_EPP6xxx.Beckhoff_EPP6xxxEK1122.A_0007_EPP6002_0002_0019.COM_TxPDO_Map_Inputs_Channel_2.Data_In[15] <-> COM TxPDO-Map Inputs Channel 2/Data In 15
//     PlcTask Inputs/GVL_iXlinker.EtherCAT_Master_EPPxxxx.Beckhoff_EPP6xxx.Beckhoff_EPP6xxxEK1122.A_0007_EPP6002_0002_0019.COM_TxPDO_Map_Inputs_Channel_2.Data_In[16] <-> COM TxPDO-Map Inputs Channel 2/Data In 16
//     PlcTask Inputs/GVL_iXlinker.EtherCAT_Master_EPPxxxx.Beckhoff_EPP6xxx.Beckhoff_EPP6xxxEK1122.A_0007_EPP6002_0002_0019.COM_TxPDO_Map_Inputs_Channel_2.Data_In[17] <-> COM TxPDO-Map Inputs Channel 2/Data In 17
//     PlcTask Inputs/GVL_iXlinker.EtherCAT_Master_EPPxxxx.Beckhoff_EPP6xxx.Beckhoff_EPP6xxxEK1122.A_0007_EPP6002_0002_0019.COM_TxPDO_Map_Inputs_Channel_2.Data_In[18] <-> COM TxPDO-Map Inputs Channel 2/Data In 18
//     PlcTask Inputs/GVL_iXlinker.EtherCAT_Master_EPPxxxx.Beckhoff_EPP6xxx.Beckhoff_EPP6xxxEK1122.A_0007_EPP6002_0002_0019.COM_TxPDO_Map_Inputs_Channel_2.Data_In[19] <-> COM TxPDO-Map Inputs Channel 2/Data In 19
//     PlcTask Inputs/GVL_iXlinker.EtherCAT_Master_EPPxxxx.Beckhoff_EPP6xxx.Beckhoff_EPP6xxxEK1122.A_0007_EPP6002_0002_0019.COM_TxPDO_Map_Inputs_Channel_2.Data_In[20] <-> COM TxPDO-Map Inputs Channel 2/Data In 20
//     PlcTask Inputs/GVL_iXlinker.EtherCAT_Master_EPPxxxx.Beckhoff_EPP6xxx.Beckhoff_EPP6xxxEK1122.A_0007_EPP6002_0002_0019.COM_TxPDO_Map_Inputs_Channel_2.Data_In[21] <-> COM TxPDO-Map Inputs Channel 2/Data In 21
//     PlcTask Outputs/GVL_iXlinker.EtherCAT_Master_EPPxxxx.Beckhoff_EPP6xxx.Beckhoff_EPP6xxxEK1122.A_0007_EPP6002_0002_0019.COM_RxPDO_Map_Outputs_Channel_1.Ctrl <-> COM RxPDO-Map Outputs Channel 1/Ctrl
//     PlcTask Outputs/GVL_iXlinker.EtherCAT_Master_EPPxxxx.Beckhoff_EPP6xxx.Beckhoff_EPP6xxxEK1122.A_0007_EPP6002_0002_0019.COM_RxPDO_Map_Outputs_Channel_2.Ctrl <-> COM RxPDO-Map Outputs Channel 2/Ctrl
//     PlcTask Outputs/GVL_iXlinker.EtherCAT_Master_EPPxxxx.Beckhoff_EPP6xxx.Beckhoff_EPP6xxxEK1122.A_0007_EPP6002_0002_0019.COM_RxPDO_Map_Outputs_Channel_1.Data_Out[0] <-> COM RxPDO-Map Outputs Channel 1/Data Out 0
//     PlcTask Outputs/GVL_iXlinker.EtherCAT_Master_EPPxxxx.Beckhoff_EPP6xxx.Beckhoff_EPP6xxxEK1122.A_0007_EPP6002_0002_0019.COM_RxPDO_Map_Outputs_Channel_1.Data_Out[1] <-> COM RxPDO-Map Outputs Channel 1/Data Out 1
//     PlcTask Outputs/GVL_iXlinker.EtherCAT_Master_EPPxxxx.Beckhoff_EPP6xxx.Beckhoff_EPP6xxxEK1122.A_0007_EPP6002_0002_0019.COM_RxPDO_Map_Outputs_Channel_1.Data_Out[2] <-> COM RxPDO-Map Outputs Channel 1/Data Out 2
//     PlcTask Outputs/GVL_iXlinker.EtherCAT_Master_EPPxxxx.Beckhoff_EPP6xxx.Beckhoff_EPP6xxxEK1122.A_0007_EPP6002_0002_0019.COM_RxPDO_Map_Outputs_Channel_1.Data_Out[3] <-> COM RxPDO-Map Outputs Channel 1/Data Out 3
//     PlcTask Outputs/GVL_iXlinker.EtherCAT_Master_EPPxxxx.Beckhoff_EPP6xxx.Beckhoff_EPP6xxxEK1122.A_0007_EPP6002_0002_0019.COM_RxPDO_Map_Outputs_Channel_1.Data_Out[4] <-> COM RxPDO-Map Outputs Channel 1/Data Out 4
//     PlcTask Outputs/GVL_iXlinker.EtherCAT_Master_EPPxxxx.Beckhoff_EPP6xxx.Beckhoff_EPP6xxxEK1122.A_0007_EPP6002_0002_0019.COM_RxPDO_Map_Outputs_Channel_1.Data_Out[5] <-> COM RxPDO-Map Outputs Channel 1/Data Out 5
//     PlcTask Outputs/GVL_iXlinker.EtherCAT_Master_EPPxxxx.Beckhoff_EPP6xxx.Beckhoff_EPP6xxxEK1122.A_0007_EPP6002_0002_0019.COM_RxPDO_Map_Outputs_Channel_1.Data_Out[6] <-> COM RxPDO-Map Outputs Channel 1/Data Out 6
//     PlcTask Outputs/GVL_iXlinker.EtherCAT_Master_EPPxxxx.Beckhoff_EPP6xxx.Beckhoff_EPP6xxxEK1122.A_0007_EPP6002_0002_0019.COM_RxPDO_Map_Outputs_Channel_1.Data_Out[7] <-> COM RxPDO-Map Outputs Channel 1/Data Out 7
//     PlcTask Outputs/GVL_iXlinker.EtherCAT_Master_EPPxxxx.Beckhoff_EPP6xxx.Beckhoff_EPP6xxxEK1122.A_0007_EPP6002_0002_0019.COM_RxPDO_Map_Outputs_Channel_1.Data_Out[8] <-> COM RxPDO-Map Outputs Channel 1/Data Out 8
//     PlcTask Outputs/GVL_iXlinker.EtherCAT_Master_EPPxxxx.Beckhoff_EPP6xxx.Beckhoff_EPP6xxxEK1122.A_0007_EPP6002_0002_0019.COM_RxPDO_Map_Outputs_Channel_1.Data_Out[9] <-> COM RxPDO-Map Outputs Channel 1/Data Out 9
//     PlcTask Outputs/GVL_iXlinker.EtherCAT_Master_EPPxxxx.Beckhoff_EPP6xxx.Beckhoff_EPP6xxxEK1122.A_0007_EPP6002_0002_0019.COM_RxPDO_Map_Outputs_Channel_1.Data_Out[10] <-> COM RxPDO-Map Outputs Channel 1/Data Out 10
//     PlcTask Outputs/GVL_iXlinker.EtherCAT_Master_EPPxxxx.Beckhoff_EPP6xxx.Beckhoff_EPP6xxxEK1122.A_0007_EPP6002_0002_0019.COM_RxPDO_Map_Outputs_Channel_1.Data_Out[11] <-> COM RxPDO-Map Outputs Channel 1/Data Out 11
//     PlcTask Outputs/GVL_iXlinker.EtherCAT_Master_EPPxxxx.Beckhoff_EPP6xxx.Beckhoff_EPP6xxxEK1122.A_0007_EPP6002_0002_0019.COM_RxPDO_Map_Outputs_Channel_1.Data_Out[12] <-> COM RxPDO-Map Outputs Channel 1/Data Out 12
//     PlcTask Outputs/GVL_iXlinker.EtherCAT_Master_EPPxxxx.Beckhoff_EPP6xxx.Beckhoff_EPP6xxxEK1122.A_0007_EPP6002_0002_0019.COM_RxPDO_Map_Outputs_Channel_1.Data_Out[13] <-> COM RxPDO-Map Outputs Channel 1/Data Out 13
//     PlcTask Outputs/GVL_iXlinker.EtherCAT_Master_EPPxxxx.Beckhoff_EPP6xxx.Beckhoff_EPP6xxxEK1122.A_0007_EPP6002_0002_0019.COM_RxPDO_Map_Outputs_Channel_1.Data_Out[14] <-> COM RxPDO-Map Outputs Channel 1/Data Out 14
//     PlcTask Outputs/GVL_iXlinker.EtherCAT_Master_EPPxxxx.Beckhoff_EPP6xxx.Beckhoff_EPP6xxxEK1122.A_0007_EPP6002_0002_0019.COM_RxPDO_Map_Outputs_Channel_1.Data_Out[15] <-> COM RxPDO-Map Outputs Channel 1/Data Out 15
//     PlcTask Outputs/GVL_iXlinker.EtherCAT_Master_EPPxxxx.Beckhoff_EPP6xxx.Beckhoff_EPP6xxxEK1122.A_0007_EPP6002_0002_0019.COM_RxPDO_Map_Outputs_Channel_1.Data_Out[16] <-> COM RxPDO-Map Outputs Channel 1/Data Out 16
//     PlcTask Outputs/GVL_iXlinker.EtherCAT_Master_EPPxxxx.Beckhoff_EPP6xxx.Beckhoff_EPP6xxxEK1122.A_0007_EPP6002_0002_0019.COM_RxPDO_Map_Outputs_Channel_1.Data_Out[17] <-> COM RxPDO-Map Outputs Channel 1/Data Out 17
//     PlcTask Outputs/GVL_iXlinker.EtherCAT_Master_EPPxxxx.Beckhoff_EPP6xxx.Beckhoff_EPP6xxxEK1122.A_0007_EPP6002_0002_0019.COM_RxPDO_Map_Outputs_Channel_1.Data_Out[18] <-> COM RxPDO-Map Outputs Channel 1/Data Out 18
//     PlcTask Outputs/GVL_iXlinker.EtherCAT_Master_EPPxxxx.Beckhoff_EPP6xxx.Beckhoff_EPP6xxxEK1122.A_0007_EPP6002_0002_0019.COM_RxPDO_Map_Outputs_Channel_1.Data_Out[19] <-> COM RxPDO-Map Outputs Channel 1/Data Out 19
//     PlcTask Outputs/GVL_iXlinker.EtherCAT_Master_EPPxxxx.Beckhoff_EPP6xxx.Beckhoff_EPP6xxxEK1122.A_0007_EPP6002_0002_0019.COM_RxPDO_Map_Outputs_Channel_1.Data_Out[20] <-> COM RxPDO-Map Outputs Channel 1/Data Out 20
//     PlcTask Outputs/GVL_iXlinker.EtherCAT_Master_EPPxxxx.Beckhoff_EPP6xxx.Beckhoff_EPP6xxxEK1122.A_0007_EPP6002_0002_0019.COM_RxPDO_Map_Outputs_Channel_1.Data_Out[21] <-> COM RxPDO-Map Outputs Channel 1/Data Out 21
//     PlcTask Outputs/GVL_iXlinker.EtherCAT_Master_EPPxxxx.Beckhoff_EPP6xxx.Beckhoff_EPP6xxxEK1122.A_0007_EPP6002_0002_0019.COM_RxPDO_Map_Outputs_Channel_2.Data_Out[0] <-> COM RxPDO-Map Outputs Channel 2/Data Out 0
//     PlcTask Outputs/GVL_iXlinker.EtherCAT_Master_EPPxxxx.Beckhoff_EPP6xxx.Beckhoff_EPP6xxxEK1122.A_0007_EPP6002_0002_0019.COM_RxPDO_Map_Outputs_Channel_2.Data_Out[1] <-> COM RxPDO-Map Outputs Channel 2/Data Out 1
//     PlcTask Outputs/GVL_iXlinker.EtherCAT_Master_EPPxxxx.Beckhoff_EPP6xxx.Beckhoff_EPP6xxxEK1122.A_0007_EPP6002_0002_0019.COM_RxPDO_Map_Outputs_Channel_2.Data_Out[2] <-> COM RxPDO-Map Outputs Channel 2/Data Out 2
//     PlcTask Outputs/GVL_iXlinker.EtherCAT_Master_EPPxxxx.Beckhoff_EPP6xxx.Beckhoff_EPP6xxxEK1122.A_0007_EPP6002_0002_0019.COM_RxPDO_Map_Outputs_Channel_2.Data_Out[3] <-> COM RxPDO-Map Outputs Channel 2/Data Out 3
//     PlcTask Outputs/GVL_iXlinker.EtherCAT_Master_EPPxxxx.Beckhoff_EPP6xxx.Beckhoff_EPP6xxxEK1122.A_0007_EPP6002_0002_0019.COM_RxPDO_Map_Outputs_Channel_2.Data_Out[4] <-> COM RxPDO-Map Outputs Channel 2/Data Out 4
//     PlcTask Outputs/GVL_iXlinker.EtherCAT_Master_EPPxxxx.Beckhoff_EPP6xxx.Beckhoff_EPP6xxxEK1122.A_0007_EPP6002_0002_0019.COM_RxPDO_Map_Outputs_Channel_2.Data_Out[5] <-> COM RxPDO-Map Outputs Channel 2/Data Out 5
//     PlcTask Outputs/GVL_iXlinker.EtherCAT_Master_EPPxxxx.Beckhoff_EPP6xxx.Beckhoff_EPP6xxxEK1122.A_0007_EPP6002_0002_0019.COM_RxPDO_Map_Outputs_Channel_2.Data_Out[6] <-> COM RxPDO-Map Outputs Channel 2/Data Out 6
//     PlcTask Outputs/GVL_iXlinker.EtherCAT_Master_EPPxxxx.Beckhoff_EPP6xxx.Beckhoff_EPP6xxxEK1122.A_0007_EPP6002_0002_0019.COM_RxPDO_Map_Outputs_Channel_2.Data_Out[7] <-> COM RxPDO-Map Outputs Channel 2/Data Out 7
//     PlcTask Outputs/GVL_iXlinker.EtherCAT_Master_EPPxxxx.Beckhoff_EPP6xxx.Beckhoff_EPP6xxxEK1122.A_0007_EPP6002_0002_0019.COM_RxPDO_Map_Outputs_Channel_2.Data_Out[8] <-> COM RxPDO-Map Outputs Channel 2/Data Out 8
//     PlcTask Outputs/GVL_iXlinker.EtherCAT_Master_EPPxxxx.Beckhoff_EPP6xxx.Beckhoff_EPP6xxxEK1122.A_0007_EPP6002_0002_0019.COM_RxPDO_Map_Outputs_Channel_2.Data_Out[9] <-> COM RxPDO-Map Outputs Channel 2/Data Out 9
//     PlcTask Outputs/GVL_iXlinker.EtherCAT_Master_EPPxxxx.Beckhoff_EPP6xxx.Beckhoff_EPP6xxxEK1122.A_0007_EPP6002_0002_0019.COM_RxPDO_Map_Outputs_Channel_2.Data_Out[10] <-> COM RxPDO-Map Outputs Channel 2/Data Out 10
//     PlcTask Outputs/GVL_iXlinker.EtherCAT_Master_EPPxxxx.Beckhoff_EPP6xxx.Beckhoff_EPP6xxxEK1122.A_0007_EPP6002_0002_0019.COM_RxPDO_Map_Outputs_Channel_2.Data_Out[11] <-> COM RxPDO-Map Outputs Channel 2/Data Out 11
//     PlcTask Outputs/GVL_iXlinker.EtherCAT_Master_EPPxxxx.Beckhoff_EPP6xxx.Beckhoff_EPP6xxxEK1122.A_0007_EPP6002_0002_0019.COM_RxPDO_Map_Outputs_Channel_2.Data_Out[12] <-> COM RxPDO-Map Outputs Channel 2/Data Out 12
//     PlcTask Outputs/GVL_iXlinker.EtherCAT_Master_EPPxxxx.Beckhoff_EPP6xxx.Beckhoff_EPP6xxxEK1122.A_0007_EPP6002_0002_0019.COM_RxPDO_Map_Outputs_Channel_2.Data_Out[13] <-> COM RxPDO-Map Outputs Channel 2/Data Out 13
//     PlcTask Outputs/GVL_iXlinker.EtherCAT_Master_EPPxxxx.Beckhoff_EPP6xxx.Beckhoff_EPP6xxxEK1122.A_0007_EPP6002_0002_0019.COM_RxPDO_Map_Outputs_Channel_2.Data_Out[14] <-> COM RxPDO-Map Outputs Channel 2/Data Out 14
//     PlcTask Outputs/GVL_iXlinker.EtherCAT_Master_EPPxxxx.Beckhoff_EPP6xxx.Beckhoff_EPP6xxxEK1122.A_0007_EPP6002_0002_0019.COM_RxPDO_Map_Outputs_Channel_2.Data_Out[15] <-> COM RxPDO-Map Outputs Channel 2/Data Out 15
//     PlcTask Outputs/GVL_iXlinker.EtherCAT_Master_EPPxxxx.Beckhoff_EPP6xxx.Beckhoff_EPP6xxxEK1122.A_0007_EPP6002_0002_0019.COM_RxPDO_Map_Outputs_Channel_2.Data_Out[16] <-> COM RxPDO-Map Outputs Channel 2/Data Out 16
//     PlcTask Outputs/GVL_iXlinker.EtherCAT_Master_EPPxxxx.Beckhoff_EPP6xxx.Beckhoff_EPP6xxxEK1122.A_0007_EPP6002_0002_0019.COM_RxPDO_Map_Outputs_Channel_2.Data_Out[17] <-> COM RxPDO-Map Outputs Channel 2/Data Out 17
//     PlcTask Outputs/GVL_iXlinker.EtherCAT_Master_EPPxxxx.Beckhoff_EPP6xxx.Beckhoff_EPP6xxxEK1122.A_0007_EPP6002_0002_0019.COM_RxPDO_Map_Outputs_Channel_2.Data_Out[18] <-> COM RxPDO-Map Outputs Channel 2/Data Out 18
//     PlcTask Outputs/GVL_iXlinker.EtherCAT_Master_EPPxxxx.Beckhoff_EPP6xxx.Beckhoff_EPP6xxxEK1122.A_0007_EPP6002_0002_0019.COM_RxPDO_Map_Outputs_Channel_2.Data_Out[19] <-> COM RxPDO-Map Outputs Channel 2/Data Out 19
//     PlcTask Outputs/GVL_iXlinker.EtherCAT_Master_EPPxxxx.Beckhoff_EPP6xxx.Beckhoff_EPP6xxxEK1122.A_0007_EPP6002_0002_0019.COM_RxPDO_Map_Outputs_Channel_2.Data_Out[20] <-> COM RxPDO-Map Outputs Channel 2/Data Out 20
//     PlcTask Outputs/GVL_iXlinker.EtherCAT_Master_EPPxxxx.Beckhoff_EPP6xxx.Beckhoff_EPP6xxxEK1122.A_0007_EPP6002_0002_0019.COM_RxPDO_Map_Outputs_Channel_2.Data_Out[21] <-> COM RxPDO-Map Outputs Channel 2/Data Out 21
//     PlcTask Inputs/GVL_iXlinker.EtherCAT_Master_EPPxxxx.Beckhoff_EPP6xxx.Beckhoff_EPP6xxxEK1122.A_0007_EPP6002_0002_0019.WcState.WcState <-> WcState/WcState
//     PlcTask Inputs/GVL_iXlinker.EtherCAT_Master_EPPxxxx.Beckhoff_EPP6xxx.Beckhoff_EPP6xxxEK1122.A_0007_EPP6002_0002_0019.WcState.InputToggle <-> WcState/InputToggle
//     PlcTask Inputs/GVL_iXlinker.EtherCAT_Master_EPPxxxx.Beckhoff_EPP6xxx.Beckhoff_EPP6xxxEK1122.A_0007_EPP6002_0002_0019.InfoData.AdsAddr <-> InfoData/AdsAddr
//     PlcTask Inputs/GVL_iXlinker.EtherCAT_Master_EPPxxxx.Beckhoff_EPP6xxx.Beckhoff_EPP6xxxEK1122.A_0007_EPP6002_0002_0019.InfoData.State <-> InfoData/State
//   PLC/PLC Instance <-> EtherCAT Master EPPxxxx/Beckhoff EPP6xxx/Beckhoff EPP6xxxEK1122/A_0008(EPP6090-0000-0017)
//     PlcTask Inputs/GVL_iXlinker.EtherCAT_Master_EPPxxxx.Beckhoff_EPP6xxx.Beckhoff_EPP6xxxEK1122.A_0008_EPP6090_0000_0017.DIS_Inputs.Status/Up <-> DIS Inputs/Status/Up
//     PlcTask Inputs/GVL_iXlinker.EtherCAT_Master_EPPxxxx.Beckhoff_EPP6xxx.Beckhoff_EPP6xxxEK1122.A_0008_EPP6090_0000_0017.DIS_Inputs.Status/Down <-> DIS Inputs/Status/Down
//     PlcTask Inputs/GVL_iXlinker.EtherCAT_Master_EPPxxxx.Beckhoff_EPP6xxx.Beckhoff_EPP6xxxEK1122.A_0008_EPP6090_0000_0017.DIS_Inputs.Status/Left <-> DIS Inputs/Status/Left
//     PlcTask Inputs/GVL_iXlinker.EtherCAT_Master_EPPxxxx.Beckhoff_EPP6xxx.Beckhoff_EPP6xxxEK1122.A_0008_EPP6090_0000_0017.DIS_Inputs.Status/Right <-> DIS Inputs/Status/Right
//     PlcTask Inputs/GVL_iXlinker.EtherCAT_Master_EPPxxxx.Beckhoff_EPP6xxx.Beckhoff_EPP6xxxEK1122.A_0008_EPP6090_0000_0017.DIS_Inputs.Status/Enter <-> DIS Inputs/Status/Enter
//     PlcTask Inputs/GVL_iXlinker.EtherCAT_Master_EPPxxxx.Beckhoff_EPP6xxx.Beckhoff_EPP6xxxEK1122.A_0008_EPP6090_0000_0017.DIS_Inputs.Status/TxPDO_Toggle <-> DIS Inputs/Status/TxPDO Toggle
//     PlcTask Outputs/GVL_iXlinker.EtherCAT_Master_EPPxxxx.Beckhoff_EPP6xxx.Beckhoff_EPP6xxxEK1122.A_0008_EPP6090_0000_0017.DIS_Outputs.Value_row[0] <-> DIS Outputs/Value row 1
//     PlcTask Outputs/GVL_iXlinker.EtherCAT_Master_EPPxxxx.Beckhoff_EPP6xxx.Beckhoff_EPP6xxxEK1122.A_0008_EPP6090_0000_0017.DIS_Outputs.Value_row[1] <-> DIS Outputs/Value row 2
//     PlcTask Inputs/GVL_iXlinker.EtherCAT_Master_EPPxxxx.Beckhoff_EPP6xxx.Beckhoff_EPP6xxxEK1122.A_0008_EPP6090_0000_0017.WcState.WcState <-> WcState/WcState
//     PlcTask Inputs/GVL_iXlinker.EtherCAT_Master_EPPxxxx.Beckhoff_EPP6xxx.Beckhoff_EPP6xxxEK1122.A_0008_EPP6090_0000_0017.WcState.InputToggle <-> WcState/InputToggle
//     PlcTask Inputs/GVL_iXlinker.EtherCAT_Master_EPPxxxx.Beckhoff_EPP6xxx.Beckhoff_EPP6xxxEK1122.A_0008_EPP6090_0000_0017.InfoData.AdsAddr <-> InfoData/AdsAddr
//     PlcTask Inputs/GVL_iXlinker.EtherCAT_Master_EPPxxxx.Beckhoff_EPP6xxx.Beckhoff_EPP6xxxEK1122.A_0008_EPP6090_0000_0017.InfoData.State <-> InfoData/State
//   PLC/PLC Instance <-> EtherCAT Master EPPxxxx/Beckhoff EPP6xxx/Beckhoff EPP6xxxEK1122/A_0009(EPP6228-0022-0016)
//     PlcTask Inputs/GVL_iXlinker.EtherCAT_Master_EPPxxxx.Beckhoff_EPP6xxx.Beckhoff_EPP6xxxEK1122.A_0009_EPP6228_0022_0016.Module_1_DeviceState_Inputs_Device.DeviceState_Inputs_Device.Device_Diag <-> Module 1 (DeviceState Inputs Device)/DeviceState Inputs Device/Device Diag
